# B&R Automation Studio project NAINV104C00R8L515F00 (part 27)

#### Local.var - Do Not Change!!!
```iecst
(*2020-09-10*)
(**)
(*Local Action, State & Status*)
VAR
	eAct : eHermesAction := HermesActIdle;
	eStat : eHermesAction := HermesActIdle;
	eMainStatus : eFBStatus := Idle;
	eStatus : eFBStatus := Idle;
	eStatus1 : eFBStatus := Idle;
	eStatus2 : eFBStatus := Idle;
	eStatus3 : eFBStatus := Idle;
	eStatus4 : eFBStatus := Idle;
	udiStatus : UDINT := 0;
	udiStatus1 : UDINT := 0;
	udiStatus2 : UDINT := 0;
	udiStatus3 : UDINT := 0;
	udiStatus4 : UDINT := 0;
	udiStatus5 : UDINT := 0;
	sStatTxt : STRING[200] := '';
	a_sStatText : ARRAY[0..50] OF STRING[200] := ['Idling','Background Starting Operations','Background Stopping Operations','Deleting Old Log File','Creating Directory','Writing Retain File','Reading Retain File','Saving Configuration',43('')];
END_VAR
(**)
(*Local Alarm*)
VAR
	tyAlmData : tyAlmDat;
	tyAlmData1 : tyAlmDat;
	tyAlmData2 : tyAlmDat;
	tyAlmData3 : tyAlmDat;
	tyAlmData4 : tyAlmDat;
	tyAlmData5 : tyAlmDat;
	tyInfoData : tyAlmDat;
	tyInfoData1 : tyAlmDat;
	tyInfoData2 : tyAlmDat;
	a_tyAlmText : ARRAY[10000..10199] OF tyAlmTxt := [(sAlmText:='Invalid Ident While Client Connecting',sRcyText:='Problem Occurred In The TCP/IP Connection. Check The Connection And Try To Reconnect.'),(sAlmText:='Setting Keep Alive Interval Time Error While Client Connecting',sRcyText:='Unable To Establish Connection Between Machine. Check For Setting And Resume Operation.'),(sAlmText:='Setting Keep Alive Idle Time Error While Client Connecting',sRcyText:='Unable To Establish Connection Between Machine. Check For Setting And Resume Operation.'),(sAlmText:='Setting Keep Alive Count Error While Client Connecting',sRcyText:='Unable To Establish Connection Between Machine. Check For Setting And Resume Operation.'),(sAlmText:='Setting Keep Alive Error While Client Connecting',sRcyText:='Unable To Establish Connection Between Machine. Check For Setting And Resume Operation.'),(sAlmText:='Setting Receive Buffer Error While Client Connecting',sRcyText:='Unable To Establish Connection Between Machine. Check For Setting And Resume Operation.'),(sAlmText:='Setting Send Buffer Error While Client Connecting',sRcyText:='Unable To Establish Connection Between Machine. Check For Setting And Resume Operation.'),(sAlmText:='Setting No Waiting Error While Client Connecting',sRcyText:='Unable To Establish Connection Between Machine. Check For Setting And Resume Operation.'),(sAlmText:='TCP Open Port Error While Client Connecting',sRcyText:='Problem Occurred In The TCP/IP Connection. Check The Connection And Try To Reconnect.'),(sAlmText:='Closing TCP Error While Client Connecting',sRcyText:='Problem Occurred In The TCP/IP Connection. Check The Connection And Try To Reconnect.'),(sAlmText:='Server Connection Failed While Client Connecting',sRcyText:='There Was A Problem Connecting To The Server. The Server May Not Exist or It is Unavailable At This Time. Check The Connection and Try Again.'),(sAlmText:='Ident In Used While Client Connecting',sRcyText:='Problem Occurred In The TCP/IP Connection. Check The Connection And Reconnect.'),(sAlmText:='Connect To Server Error While Client Connecting',sRcyText:='There Was A Problem Connecting To The Server. The Server May Not Exist or It is Unavailable At This Time. Check The Connection and Try Again.'),(sAlmText:='US Hermes Connection Lost',sRcyText:='Please Check Network Connection.'),(sAlmText:='Invalid Ident While Receiving Data',sRcyText:='Problem Occurred In The TCP/IP Connection. Check The Connection And Try To Reconnect.'),(sAlmText:='TCP Receive Data Error While Receiving Data',sRcyText:='Problem Occurred In The TCP/IP Connection. Check The Connection And Try To Reconnect.'),(sAlmText:='Receive ServiceDescription While Upstream In Not Connected State',sRcyText:='Receive Illegal Message.'),(sAlmText:='Receive BoardAvailable While Upstream In Not Connected State',sRcyText:='Receive Illegal Message.'),(sAlmText:='Receive RevokeBoardAvailable While Upstream In Not Connected State',sRcyText:='Receive Illegal Message.'),(sAlmText:='Receive MachineReady While Upstream In Not Connected State',sRcyText:='Receive Illegal Message.'),(sAlmText:='Receive RevokeMachineReady While Upstream In Not Connected State',sRcyText:='Receive Illegal Message.'),(sAlmText:='Receive StartTransport While Upstream In Not Connected State',sRcyText:='Receive Illegal Message.'),(sAlmText:='Receive StopTransport While Upstream In Not Connected State',sRcyText:='Receive Illegal Message.'),(sAlmText:='Receive TransportFinished While Upstream In Not Connected State',sRcyText:='Receive Illegal Message.'),(sAlmText:='Receive BoardForecast While Upstream In Not Connected State',sRcyText:='Receive Illegal Message.'),(sAlmText:='Receive BoardAvailable While Upstream In Service Description State',sRcyText:='Receive Illegal Message.'),(sAlmText:='Receive RevokeBoardAvailable While Upstream In Service Description State',sRcyText:='Receive Illegal Message.'),(sAlmText:='Receive MachineReady While Upstream In Service Description State',sRcyText:='Receive Illegal Message.'),(sAlmText:='Receive RevokeMachineReady While Upstream In Service Description State',sRcyText:='Receive Illegal Message.'),(sAlmText:='Receive StartTransport While Upstream In Service Description State',sRcyText:='Receive Illegal Message.'),(sAlmText:='Receive StopTransport While Upstream In Service Description State',sRcyText:='Receive Illegal Message.'),(sAlmText:='Receive TransportFinished While Upstream In Service Description State',sRcyText:='Receive Illegal Message.'),(sAlmText:='Receive BoardForecast While Upstream In Service Description State',sRcyText:='Receive Illegal Message.'),(sAlmText:='Receive ServiceDescription While Upstream In Not Available Not Ready State',sRcyText:='Receive Illegal Message.'),(sAlmText:='Receive RevokeBoardAvailable While Upstream In Not Available Not Ready State',sRcyText:='Receive Illegal Message.'),(sAlmText:='Receive MachineReady While Upstream In Not Available Not Ready State',sRcyText:='Receive Illegal Message.'),(sAlmText:='Receive RevokeMachineReady While Upstream In Not Available Not Ready State',sRcyText:='Receive Illegal Message.'),(sAlmText:='Receive StartTransport While Upstream In Not Available Not Ready State',sRcyText:='Receive Illegal Message.'),(sAlmText:='Receive StopTransport While Upstream In Not Available Not Ready State',sRcyText:='Receive Illegal Message.'),(sAlmText:='Receive TransportFinished While Upstream In Not Available Not Ready State',sRcyText:='Receive Illegal Message.'),(sAlmText:='Receive ServiceDescription While Upstream In Board Available State',sRcyText:='Receive Illegal Message.'),(sAlmText:='Receive BoardAvailable While Upstream In Board Available State',sRcyText:='Receive Illegal Message.'),(sAlmText:='Receive MachineReady While Upstream In Board Available State',sRcyText:='Receive Illegal Message.'),(sAlmText:='Receive RevokeMachineReady While Upstream In Board Available State',sRcyText:='Receive Illegal Message.'),(sAlmText:='Receive StartTransport While Upstream In Board Available State',sRcyText:='Receive Illegal Message.'),(sAlmText:='Receive StopTransport While Upstream In Board Available State',sRcyText:='Receive Illegal Message.'),(sAlmText:='Receive TransportFinished While Upstream In Board Available State',sRcyText:='Receive Illegal Message.'),(sAlmText:='Receive BoardForecast While Upstream In Board Available State',sRcyText:='Receive Illegal Message.'),(sAlmText:='Receive ServiceDescription While Upstream In Machine Ready State',sRcyText:='Receive Illegal Message.'),(sAlmText:='Receive RevokeBoardAvailable While Upstream In Machine Ready State',sRcyText:='Receive Illegal Message.'),(sAlmText:='Receive MachineReady While Upstream In Machine Ready State',sRcyText:='Receive Illegal Message.'),(sAlmText:='Receive RevokeMachineReady While Upstream In Machine Ready State',sRcyText:='Receive Illegal Message.'),(sAlmText:='Receive StartTransport While Upstream In Machine Ready State',sRcyText:='Receive Illegal Message.'),(sAlmText:='Receive StopTransport While Upstream In Machine Ready State',sRcyText:='Receive Illegal Message.'),(sAlmText:='Receive TransportFinished While Upstream In Machine Ready State',sRcyText:='Receive Illegal Message.'),(sAlmText:='Receive ServiceDescription While Upstream In Available And Ready State',sRcyText:='Receive Illegal Message.'),(sAlmText:='Receive BoardAvailable While Upstream In Available And Ready State',sRcyText:='Receive Illegal Message.'),(sAlmText:='Receive MachineReady While Upstream In Available And Ready State',sRcyText:='Receive Illegal Message.'),(sAlmText:='Receive RevokeMachineReady While Upstream In Available And Ready State',sRcyText:='Receive Illegal Message.'),(sAlmText:='Receive StartTransport While Upstream In Available And Ready State',sRcyText:='Receive Illegal Message.'),(sAlmText:='Receive StopTransport While Upstream In Available And Ready State',sRcyText:='Receive Illegal Message.'),(sAlmText:='Receive TransportFinished While Upstream In Available And Ready State',sRcyText:='Receive Illegal Message.'),(sAlmText:='Receive BoardForecast While Upstream In Available And Ready State',sRcyText:='Receive Illegal Message.'),(sAlmText:='Receive ServiceDescription While Upstream In Transporting State',sRcyText:='Receive Illegal Message.'),(sAlmText:='Receive Twice Board Available While Upstream In Transporting State',sRcyText:='Receive Illegal Message.'),(sAlmText:='Receive RevokeBoardAvailable Without BoardAvailable While Upstream In Transporting State',sRcyText:='Receive Illegal Message.'),(sAlmText:='Receive MachineReady While Upstream In Transporting State',sRcyText:='Receive Illegal Message.'),(sAlmText:='Receive RevokeMachineReady While Upstream In Transporting State',sRcyText:='Receive Illegal Message.'),(sAlmText:='Receive StartTransport While Upstream In Transporting State',sRcyText:='Receive Illegal Message.'),(sAlmText:='Receive StopTransport While Upstream In Transporting State',sRcyText:='Receive Illegal Message.'),(sAlmText:='Receive ServiceDescription While Upstream In Transport Finished State',sRcyText:='Receive Illegal Message.'),(sAlmText:='Receive BoardAvailable While Upstream In Transport Finished State',sRcyText:='Receive Illegal Message.'),(sAlmText:='Receive RevokeBoardAvailable While UpstreamWhile Upstream In Transport Finished State',sRcyText:='Receive Illegal Message.'),(sAlmText:='Receive MachineReady While Upstream In Transport Finished State',sRcyText:='Receive Illegal Message.'),(sAlmText:='Receive RevokeMachineReady While Upstream In Transport Finished State',sRcyText:='Receive Illegal Message.'),(sAlmText:='Receive StartTransport While Upstream In Transport Finished State',sRcyText:='Receive Illegal Message.'),(sAlmText:='Receive TransportFinished While Upstream In Transport Finished State',sRcyText:='Receive Illegal Message.'),(sAlmText:='Receive StopTransport While Upstream In Transport Finished State',sRcyText:='Receive Illegal Message.'),(sAlmText:='Receive BoardForecast While Upstream In Transport Finished State',sRcyText:='Receive Illegal Message.'),(sAlmText:='Receive ServiceDescription While Upstream In Transport Stopped State',sRcyText:='Receive Illegal Message.'),(sAlmText:='Receive Twice Board Available While Upstream In Transport Stopped State',sRcyText:='Receive Illegal Message.'),(sAlmText:='Receive RevokeBoardAvailable Without BoardAvailable While Upstream In Transport Stopped State',sRcyText:='Receive Illegal Message.'),(sAlmText:='Receive MachineReady While Upstream In Transport Stopped State',sRcyText:='Receive Illegal Message.'),(sAlmText:='Receive RevokeMachineReady While Upstream In Transport Stopped State',sRcyText:='Receive Illegal Message.'),(sAlmText:='Receive StartTransport While Upstream In Transport Stopped State',sRcyText:='Receive Illegal Message.'),(sAlmText:='Receive StopTransport While Upstream In Transport Stopped State',sRcyText:='Receive Illegal Message.'),(sAlmText:='LaneId Mismatch While Checking Service Description',sRcyText:='The LaneId Value Does Not Match. Change The Value And Resend The Value.'),(sAlmText:='MachineId Missing While Checking Service Description',sRcyText:='Missing Input Value For MachineId. Fill Up The Value And Resend.'),(sAlmText:='LandId Out Of Range While Checking Service Description',sRcyText:='LaneId Does Not Fall Within The Expected Range.'),(sAlmText:='LandId Missing While Checking Service Description',sRcyText:='Missing Input Value For LaneId. Fill Up The Value And Resend.'),(sAlmText:='Version Missing While Checking Service Description',sRcyText:='Missing Input Value For Version. Fill Up The Value And Resend.'),(sAlmText:='SupportedFeatures Missing While Checking Service Description',sRcyText:='Missing Input Value For SupportedFeatures. Fill Up The Value And Resend.'),(sAlmText:='NotificationCode Out Of Range While Checking Notification',sRcyText:='NotificationCode Does Not Fall Within The Expected Range.'),(sAlmText:='NotificationCode Missing While Checking Notification',sRcyText:='Missing Input Value For NotificationCode. Fill Up The Value And Resend.'),(sAlmText:='Severity Missing While Checking Notification',sRcyText:='Missing Input Value For Severity. Fill Up The Value And Resend.'),(sAlmText:='Description Missing While Checking Notification',sRcyText:='Missing Input Value For Description. Fill Up The Value And Resend.'),(sAlmText:='BoardId Missing While Checking Board Available',sRcyText:='Missing Input Value For BoardId. Fill Up The Value And Resend.'),(sAlmText:='BoardIdCreatedBy Missing While Checking Board Available',sRcyText:='Missing Input Value For BoardIdCreatedBy. Fill Up The Value And Resend.'),(sAlmText:='FailedBoard Missing While Checking Board Available',sRcyText:='Missing Input Value For FailedBoard. Fill Up The Value And Resend.'),(sAlmText:='FlippedBoard Missing While Checking Board Available',sRcyText:='Missing Input Value For FlippedBoard. Fill Up The Value And Resend.'),(sAlmText:='TransferState Missing While Checking Transport Finished',sRcyText:='Missing Input Value For TransferState. Fill Up The Value And Resend.'),(sAlmText:='BoardId Missing While Checking Transport Finished',sRcyText:='Missing Input Value For BoardId. Fill Up The Value And Resend.'),(sAlmText:='FailedBoard Missing While Checking Board Forecast',sRcyText:='Missing Input Value For FailedBoard. Fill Up The Value And Resend.'),(sAlmText:='FlippedBoard Missing While Checking Board Forecast',sRcyText:='Missing Input Value For FlippedBoard. Fill Up The Value And Resend.'),(sAlmText:='BoardId Mismatch While Checking Start Transport & Transport Finished',sRcyText:='The BoardId Value Does Not Match. Change The Value And Resend The Value.'),(sAlmText:='BoardId Missing While Checking Start Transport & Transport Finished',sRcyText:='Missing Input Value For BoardId. Fill Up The Value And Resend.'),(sAlmText:='Service Description Interchange Time Out',sRcyText:='Timeout Expired Before Operation Completed. Reset And Resume Operation.'),(sAlmText:='Transport Time Out',sRcyText:='Timeout Expired Before Operation Completed. Reset And Resume Operation.'),(sAlmText:='Input First Slot Is Invalid',sRcyText:='Invalid Input Value.'),(sAlmText:='Input Last Slot Is Invalid',sRcyText:='Invalid Input Value.'),(sAlmText:='Input Pitch Is Invalid',sRcyText:='Invalid Input Value.'),(sAlmText:='Input Slot To Slot Distance Is Invalid',sRcyText:='Invalid Input Value.'),(sAlmText:='Input Total Slot Is Invalid',sRcyText:='Invalid Input Value.'),(sAlmText:='Input Thickness Is Invalid',sRcyText:='Invalid Input Value.'),(sAlmText:='Input Top Clearance Height Is Invalid',sRcyText:='Invalid Input Value.'),(sAlmText:='Input Bottom Clearance Height Is Invalid',sRcyText:='Invalid Input Value.'),(sAlmText:='Recipe First Slot Value & Board Available Data Not Match With Same Product Type Id',sRcyText:='The Recipe First Slot Value & Board Available Data Value Does Not Match With Product Type ID. Change The Value And Resend The Value.'),(sAlmText:='Recipe Last Slot Value & Board Available Data Not Match With Same Product Type Id',sRcyText:='The Recipe Last Slot Value & Board Available Data Value Does Not Match With Product Type ID. Change The Value And Resend The Value.'),(sAlmText:='Recipe Pitch Value & Board Available Data Not Match With Same Product Type Id',sRcyText:='The Recipe Pitch Value & Board Available Data Value Does Not Match With Product Type ID. Change The Value And Resend The Value.'),(sAlmText:='Width Different With Same Product Type Id',sRcyText:='Width Does Not Match With Product Type ID. Change The Value And Resend The Value.'),(sAlmText:='Input First Slot Is Invalid',sRcyText:='Invalid Input Value.'),(sAlmText:='Input Last Slot Is Invalid',sRcyText:='Invalid Input Value.'),(sAlmText:='Input Pitch Is Invalid',sRcyText:='Invalid Input Value.'),(sAlmText:='Input Slot To Slot Distance Is Invalid',sRcyText:='Invalid Input Value.'),(sAlmText:='Input Total Slot Is Invalid',sRcyText:='Invalid Input Value.'),(sAlmText:='Input Thickness Is Invalid',sRcyText:='Invalid Input Value.'),(sAlmText:='Input Top Clearance Height Is Invalid',sRcyText:='Invalid Input Value.'),(sAlmText:='Input Bottom Clearance Height Is Invalid',sRcyText:='Invalid Input Value.'),(sAlmText:='Recipe First Slot Value & Board Available Data Not Match With Same Product Type Id',sRcyText:='The Recipe First Slot Value & Board Available Data Value Does Not Match With Product Type ID. Change The Value And Resend The Value.'),(sAlmText:='Recipe Last Slot Value & Board Available Data Not Match With Same Product Type Id',sRcyText:='The Recipe Last Slot Value & Board Available Data Value Does Not Match With Product Type ID. Change The Value And Resend The Value.'),(sAlmText:='Recipe Pitch Value & Board Available Data Not Match With Same Product Type Id',sRcyText:='The Recipe Pitch Value & Board Available Data Value Does Not Match With Product Type ID. Change The Value And Resend The Value.'),(sAlmText:='Width Different With Same Product Type Id',sRcyText:='Width Does Not Match With Product Type ID. Change The Value And Resend The Value.'),(sAlmText:='Check Alive Time Out',sRcyText:='Timeout Expired Before Operation Completed. Reset And Resume Operation.'),(sAlmText:='Waiting Check Alive Time Out',sRcyText:='Timeout Expired Before Operation Completed. Reset And Resume Operation.'),(sAlmText:='Check Alive Id Mismatch',sRcyText:='The Check Alive Id Value Does Not Match. Change The Value And Resend The Value.'),(sAlmText:='Board Available Request To Send From Upstream Hermes',sRcyText:='Sending Illegal Message.'),(sAlmText:='Revoke Board Available Request To Send From Upstream Hermes',sRcyText:='Sending Illegal Message.'),(sAlmText:='Transport Finished Request To Send From Upstream Hermes',sRcyText:='Sending Illegal Message.'),(sAlmText:='Set Configuration Request To Send From Upstream Hermes',sRcyText:='Sending Illegal Message.'),(sAlmText:='Get Configuration Request To Send From Upstream Hermes',sRcyText:='Sending Illegal Message.'),(sAlmText:='Current Configuration Request To Send From Upstream Hermes',sRcyText:='Sending Illegal Message.'),(sAlmText:='Board Forecast Request To Send From Upstream Hermes',sRcyText:='Sending Illegal Message.'),(sAlmText:='Send Board Info Request To Send From Upstream Hermes',sRcyText:='Sending Illegal Message.'),(sAlmText:='Invalid Ident While Sending Data',sRcyText:='Invalid Ident Value.'),(sAlmText:='TCP Retry Send Data Error While Sending Data',sRcyText:='Problem Occurred In The TCP/IP Connection. Check The Connection And Try To Reconnect.'),(sAlmText:='TCP Send Data Error',sRcyText:='Problem Occurred In The TCP/IP Connection. Check The Connection And Try To Reconnect.'),(sAlmText:='Invalid Ident While Closing TCP',sRcyText:='Invalid Ident Value.'),(sAlmText:='Closing TCP Error',sRcyText:='Problem Occurred In The TCP/IP Connection. Check The Connection And Try To Reconnect.'),(sAlmText:='File Open Error While Writing Log',sRcyText:='An Error Was Encountered While Trying To Open File. Please Contact Nutek For A Possible Solution.'),(sAlmText:='File Create Error While Writing Log',sRcyText:='An Error Was Encountered While Trying To Create File. Please Contact Nutek For A Possible Solution.'),(sAlmText:='Get File Info Error While Writing Log',sRcyText:='An Error Was Encountered While Getting File Info. Please Contact Nutek For A Possible Solution.'),(sAlmText:='File Write Error While Writing Log',sRcyText:='An Error Was Encountered While Trying To Write File. Please Contact Nutek For A Possible Solution.'),(sAlmText:='File Close Error While Writing Log',sRcyText:='An Error Was Encountered While Trying To Close File. Please Contact Nutek For A Possible Solution.'),(sAlmText:='Directory Does Not Exist While Writing Log',sRcyText:='The Directory Does Not Exist.Please Contact Nutek For A Possible Solution.'),(sAlmText:='Get Directory Info Error While Deleting Old Log',sRcyText:='An Error Was Encountered While Getting Directory Info. Please Contact Nutek For A Possible Solution.'),(sAlmText:='Directory Read Error While Deleting Old Log',sRcyText:='An Error Was Encountered While Reading Directory. Please Contact Nutek For A Possible Solution.'),(sAlmText:='File Delete Error While Deleting Old Log',sRcyText:='An Error Was Encountered While Trying To Delete File. Please Contact Nutek For A Possible Solution.'),(sAlmText:='Board Jam At Sensor After Transfer Interrupted',sRcyText:='Push Back Board To Upstream Machine'),(sAlmText:='Product Type Id Not Receive From Upstream',sRcyText:='Check Upstream Machine Whether Product Type Id Is Used.'),10((0)),(sAlmText:='New Recipe Not Found In Product Recipe List',sRcyText:='Create New Recipe In Product Setting.'),30((0))];
END_VAR
(**)
(*Local Output*)
VAR
	a_tyXMLTableDataBrdAvl : ARRAY[0..200] OF tyXMLTableDat;
	iXMLTableDataBrdAvlTtlIdx : INT;
	bConnected : BOOL;
	bHandshakeDone : BOOL;
	bBoardChkReq : BOOL;
	bAccDataReq : BOOL;
	bProcessBoardForecastId : BOOL;
	bBFAccDataReq : BOOL;
	bOverWriteSlt : BOOL;
	bBFOverWriteSlt : BOOL;
	bBFOverWriteWidth : BOOL;
	bOverWriteWidth : BOOL;
	sReqRecipeNm : STRING[254];
	diReqWidthInUM : DINT;
	diReqMinSltValue : DINT;
	diReqMaxSltValue : DINT;
	diReqPitch : DINT;
	bNotAvlNotRdy : BOOL;
	bUSRdy : BOOL;
	bDSRdy : BOOL;
	bUSGdRdy : BOOL;
	bDSGdRdy : BOOL;
	iAction : INT;
	bTransporting : BOOL;
	bStopTransport : BOOL;
	tyBoardAvailableRcv : tyHermesBoardAvailable;
	tyBoardAvailableReq : tyHermesBoardAvailable;
	bBlkUS : BOOL;
	bBABlkUS : BOOL;
	bBFBlkUS : BOOL;
	bManuallInsertLastZone : BOOL;
	bReverseRcvBlkUS : BOOL;
	sInternalSnd : STRING[65535];
	bRcvBoardInfoOk : BOOL;
	bRcvBoardInfoIncompl : BOOL;
	tySendBoardInfoAcc : tyHermesSendBoardInfo;
END_VAR
(**)
(*Local Input*)
VAR
	udiRstErr : UDINT := 0;
	bPrep : BOOL := TRUE;
	bEn : BOOL := TRUE;
	bDis : BOOL := FALSE;
	tyParam : tyHermesUSParam := (tSndAlive:=T#30s,tRcvAlive:=T#60s,iLaneID:=1,sHostAddress:='192.168.0.200',uiHostPort:=5000);
	sIPAddr : STRING[15] := '192.168.0.100';
	tyDTStructure : DTStructure := (year:=2019,month:=01,day:=05,wday:=05,hour:=21,minute:=28,second:=30,millisec:=123,microsec:=456);
	dtCurrDT : DATE_AND_TIME := DT#2019-02-23-12:30:50;
	bRdyRcv : BOOL := FALSE;
	bRdyTransport : BOOL := FALSE;
	bRcvCompl : BOOL := FALSE;
	bRcvInCompl : BOOL := FALSE;
	bRcvNotStart : BOOL := FALSE;
	bBAWidthEn : BOOL := TRUE; (*Board Available Check Width*)
	bBASltEn : BOOL := FALSE; (*Board Available Check Slot*)
	bBFWidthEn : BOOL := TRUE; (*Board Forecast Check Width*)
	bBFSltEn : BOOL := FALSE; (*Board Forecast Check Slot*)
	sMcId : STRING[80] := '';
	sInterfaceId : STRING[80] := '';
	sVersion : STRING[7] := '1.0.2';
	eFailedBoard : eHermesFailedBoard := HermesUnknownBoard;
	sRecipeNm : STRING[254] := '';
	diWidthInUM : DINT := 0;
	diMinSltValue : DINT := 0;
	diMaxSltValue : DINT := 0;
	diPitch : DINT := 0;
	diTtlSlt : DINT := 0;
	diSltToSltInUM : DINT := 0;
	udiSndBffrSize : UDINT := 65536;
	udiRcvBffrSize : UDINT := 65536;
	udiAliveIdleTimeInSec : UDINT := 5;
	tConnTimeOut : TIME := T#30s;
	diTransferInTO : DINT := 30000;
	bOpsRun : BOOL := FALSE;
	bInterruptSen : BOOL := FALSE;
	udiFileKeepDay : UDINT := 30;
	sProgNm : STRING[15] := 'USHermes';
	bNtSettingsLoadDone : BOOL := TRUE;
	bAccDataRdy : BOOL := FALSE;
	sRmtMcId : STRING[80];
	bRmtPrep : BOOL := FALSE;
	bRmtEn : BOOL := FALSE;
	bAccNewRcpCond : BOOL;
	sInfoMsg : STRING[200];
	sInfoMsg1 : STRING[200];
	sInfoMsg2 : STRING[200];
	bInternalUse : BOOL;
	sInternalRcv : STRING[65535];
	a_tyProdRcpList : ARRAY[1..c_udiProdRcpMax] OF tyProdRcpParam;
	tyProdRcpCurrRcp : tyProdRcpParam;
	bMcParamMnlAccData : BOOL;
	bUIAccData : BOOL;
END_VAR
(**)
(*Local*)
VAR
	bRstErr : BOOL;
	udiRstErrOld : UDINT;
	bInitDone : BOOL;
	bInitialDone : BOOL;
	bRun : BOOL;
	bStop : BOOL;
	bRstConnection : BOOL;
	bRstState : BOOL;
	udiTCPIdent : UDINT;
	udiXMLTableWriteIdx : UDINT;
	udiMsgSendBffr : UDINT;
	udiSndMsgLen : UDINT;
	sSnd : STRING[65535];
	sRcv : STRING[65535];
	a_tyXMLTableDataRcv : ARRAY[0..200] OF tyXMLTableDat;
	a_tyXMLTableDataSnd : ARRAY[0..200] OF tyXMLTableDat;
	a_eMsgSend : ARRAY[0..50] OF eHermesMsgType;
	tyMsgTypeRcv : tyHermesMsgType;
	tyCheckAliveSnd : tyHermesCheckAlive;
	tyCheckAlivePingSnd : tyHermesCheckAlive;
	tyCheckAlivePongSnd : tyHermesCheckAlive;
	tyCheckAliveRcv : tyHermesCheckAlive;
	tyCheckAlivePingRcv : tyHermesCheckAlive;
	tyCheckAlivePongRcv : tyHermesCheckAlive;
	tyServiceDescriptionSnd : tyHermesServiceDescription;
	tyServiceDescriptionRcv : tyHermesServiceDescription;
	tyNotificationSnd : tyHermesNotification;
	tyNotificationRcv : tyHermesNotification;
	tyBoardAvailableDummy : tyHermesBoardAvailable;
	tyBoardArrivedInfo : tyHermesBoardAvailable;
	tyMachineReady : tyHermesMachineReady;
	tyStartTransport : tyHermesStartTransport;
	tyStopTransport : tyHermesStopTransport;
	tyTransportFinished : tyHermesTransportFinished;
	tySetConfiguration : tyHermesSetConfiguration;
	tyCurrentConfiguration : tyHermesCurrentConfiguration;
	tyBoardForecastRcv : tyHermesBoardForecast;
	tyBoardForecastAcc : tyHermesBoardForecast;
	tyQueryBoardInfo : tyHermesQueryBoardInfo;
	tySendBoardInfoRcv : tyHermesSendBoardInfo;
	tyCommandRcv : tyHermesCommand;
	tyCommandSnd : tyHermesCommand;
	fbClntConnect : fbTCPClntConnect;
	fbRcv : fbTCPRcv;
	fbSend : fbTCPSnd;
	fbClose : fbTCPClose;
	fbParseXMLTable : fbHermesParseXMLTable;
	fbCheckAlive : fbHermesCheckAlive;
	fbCheckAliveSendPing : fbHermesCheckAliveSendPing;
	fbCheckAliveRcvPing : fbHermesCheckAliveRcvPing;
	fbSequenceUS : fbHermesSequenceUS;
	fbSequenceTO : fbHermesSequenceTO;
	fbGetSlt : fbHermesGetSlt;
	eStatOld : eHermesAction := HermesActIdle;
	tyParamOld : tyHermesUSParam;
	udiLogCntr : UDINT := 1;
	udiWriteLogCntr : UDINT := 1;
	a_sLogList : ARRAY[1..10] OF STRING[65535];
	sDT : STRING[80];
	dtCurrDTTemp : DATE_AND_TIME;
	fbFileAppend1 : fbFileFullAppend;
	fbFileOldDel1 : fbFileOldDel;
	iWriteLogStep : INT := 0;
	i : INT;
	usiBFAccDataStep : USINT;
	usiAccDataStep : USINT;
	bFeatureBoardForecast : BOOL;
	bAccDataMnl : BOOL;
	bStopTransportSnd : BOOL;
	tyCommandParam : tyHermesCommandParam;
	a_usiHermesCommandIdx : ARRAY[0..7] OF USINT;
	udiModuleNum : UDINT := 3101;
	bReplyMcRdyId : BOOL;
	bBrdForecastRcv : BOOL;
END_VAR
(*Reverse Trigger*)
VAR
	bProcessRouteMachine : BOOL;
	bTriggerRouteMachine : BOOL;
	bProcessRouteReversal : BOOL;
	bTriggerRouteReversal : BOOL;
	iGotoLane : INT;
	bManualRmvBrdCond : BOOL;
	bReverseDSSndBfWBrdID : BOOL;
	bTriggerUpdateRoute : BOOL;
	bNotifyRstReverseRcvGate : BOOL;
	fbRstReverseRcvGate : TON;
	fbRstReverseDSSndBF : TON;
	usidx : USINT;
	iMinDis : INT;
	bSwitchtoReverseReceive : BOOL;
	fbRstSndBF : TON;
	bStopTransportSent : BOOL;
	bBoardAvailableRcved : BOOL;
END_VAR
(*Insert your comment here.*)
VAR
	bManualRmvRoute : BOOL;
	bReturnRoute : BOOL;
	bNomRouteEn : BOOL;
	bProcessRouteEn : BOOL;
	bReverseReceiveRoute : BOOL;
	bReceiveReverseUSMcRdy : BOOL;
	bReverseSentRoute : BOOL;
END_VAR
(*QueryBoard Info*)
VAR
	sUITopBarcode : STRING[254];
	sUIBottomBarcode : STRING[254];
END_VAR
```

### USHermes2.var - Change By Project
```iecst
(*2020-09-10*)
(**)
(*Action & State & Status*)
VAR
	p_USHermes2Stat : UDINT;
	p_USHermes2Status : UDINT;
	p_USHermes2StatTxt : UDINT;
END_VAR
(**)
(*Alarm*)
VAR
	p_USHermes2AlmData : UDINT;
	p_USHermes2AlmData1 : UDINT;
	p_USHermes2AlmData2 : UDINT;
	p_USHermes2AlmData3 : UDINT;
	p_USHermes2AlmData4 : UDINT;
	p_USHermes2AlmData5 : UDINT;
	p_USHermes2InfoData : UDINT;
END_VAR
(**)
(*Output*)
VAR
	p_USHermes2TableDataBrdAvl : UDINT;
	p_USHermes2TableDataBrdAvlTtlIdx : UDINT;
	p_USHermes2Connected : UDINT;
	p_USHermes2HandshakeDone : UDINT;
	p_USHermes2AccDataReq : UDINT;
	p_USHermes2OverWriteSlt : UDINT;
	p_USHermes2OverWriteWidth : UDINT;
	p_USHermes2ReqRecipeNm : UDINT;
	p_USHermes2ReqWidthInUM : UDINT;
	p_USHermes2ReqMinSltValue : UDINT;
	p_USHermes2ReqMaxSltValue : UDINT;
	p_USHermes2ReqPitch : UDINT;
	p_USHermes2USRdy : UDINT;
	p_USHermes2DSRdy : UDINT;
	p_USHermes2USGdRdy : UDINT;
	p_USHermes2DSGdRdy : UDINT;
	p_USHermes2Transporting : UDINT;
	p_USHermes2StopTransport : UDINT;
	p_USHermes2BlkUS : UDINT;
	p_USHermes2InternalSnd : UDINT;
	p_USHermes2AccDataMnl : UDINT;
	p_USHermes2tyBoardAvailable : UDINT;
	p_USHermes2CommandParam : UDINT;
	p_USHermes2ReverseDSSendBFId : UDINT;
	p_USHermes2ProcessRouteTrigger : UDINT;
	p_USHermes2SwitchtoReverseRcv : UDINT;
	p_USHermes2StopTransportSnd : UDINT;
	p_USHermes2RcvBoardInfoOk : UDINT;
	p_USHermes2RcvbBoardInfoIncompl : UDINT;
	p_USHermes2BoardInfoData : UDINT;
	p_USHermes2BoardArrivedData : UDINT;
	p_USHermes2BrdForecastRcv : UDINT;
	p_USHermes2BoardAvailableRcved : UDINT;
	p_USHermes2StopTransportSent : UDINT;
	p_USHermes2StopTransportSentMsg : UDINT;
	p_USHermes2BrdForecast : UDINT;
END_VAR
```

### Program Logical/Hermes/USHermes2 (IEC) - 1.00.0 - NtHermes v5.00.0 , NtTCP v5.00.0 , NtMessage v5.00.0

#### InputRef.var
```iecst
(*2019-06-28*)
(**)
(*General*)
VAR
	p_eAct : REFERENCE TO eHermesAction;
	p_udiRstErr : REFERENCE TO UDINT;
	p_bPrep : REFERENCE TO BOOL;
	p_bEn : REFERENCE TO BOOL;
	p_bDis : REFERENCE TO BOOL;
END_VAR
(**)
(*Configuration*)
VAR
	p_tyParam : REFERENCE TO tyHermesUSParam;
	p_sIPAddr : REFERENCE TO STRING[15];
	p_tyDTStructure : REFERENCE TO DTStructure;
	p_dtCurrDT : REFERENCE TO DATE_AND_TIME;
END_VAR
(**)
(*Input*)
VAR
	p_bRdyRcv : REFERENCE TO BOOL;
	p_bRdyTransport : REFERENCE TO BOOL;
	p_bRcvCompl : REFERENCE TO BOOL;
	p_bRcvIncompl : REFERENCE TO BOOL;
	p_bRcvNotStart : REFERENCE TO BOOL;
	p_bBAWidthEn : REFERENCE TO BOOL; (*Board Available Check Width*)
	p_bBASltEn : REFERENCE TO BOOL; (*Board Available Check Slot*)
	p_bBFWidthEn : REFERENCE TO BOOL; (*Board Forecast Check Width*)
	p_bBFSltEn : REFERENCE TO BOOL; (*Board Forecast Check Slot*)
	p_sMcId : REFERENCE TO STRING[80];
	p_sInterfaceId : REFERENCE TO STRING[80];
	p_sVersion : REFERENCE TO STRING[7];
	p_eFailedBoard : REFERENCE TO eHermesFailedBoard;
	p_eFlippedBoard : REFERENCE TO eHermesFlippedBoard;
	p_sRecipeNm : REFERENCE TO STRING[254];
	p_diWidthInUM : REFERENCE TO DINT;
	p_diMinSltValue : REFERENCE TO DINT;
	p_diMaxSltValue : REFERENCE TO DINT;
	p_diPitch : REFERENCE TO DINT;
	p_diTtlSlt : REFERENCE TO DINT;
	p_diSltToSltInUM : REFERENCE TO DINT;
	p_udiSndBffrSize : REFERENCE TO UDINT;
	p_udiRcvBffrSize : REFERENCE TO UDINT;
	p_udiAliveIdleTimeInSec : REFERENCE TO UDINT;
	p_tConnTimeOut : REFERENCE TO TIME;
	p_diTransferInTO : REFERENCE TO DINT;
	p_bOpsRun : REFERENCE TO BOOL;
	p_bInterruptSen : REFERENCE TO BOOL;
	p_udiFileKeepDay : REFERENCE TO UDINT;
	p_sProgNm : REFERENCE TO STRING[15];
	p_bNtSettingsLoadDone : REFERENCE TO BOOL;
	p_bAccDataRdy : REFERENCE TO BOOL;
	p_sRmtMcId : REFERENCE TO STRING[80];
	p_bRmtPrep : REFERENCE TO BOOL;
	p_bRmtEn : REFERENCE TO BOOL;
	p_bSvyPrep : REFERENCE TO BOOL;
	p_bSvyEn : REFERENCE TO BOOL;
	p_bAccNewRcpCond : REFERENCE TO BOOL;
	p_sInfoMsg : REFERENCE TO STRING[200];
	p_sInfoMsg1 : REFERENCE TO STRING[200];
	p_sInfoMsg2 : REFERENCE TO STRING[200];
	p_bInternalUse : REFERENCE TO BOOL;
	p_sInternalRcv : REFERENCE TO STRING[65535];
	p_tyCommand : REFERENCE TO tyHermesCommand;
	pa_tyProdRcpList : REFERENCE TO ARRAY[1..c_udiProdRcpMax] OF tyProdRcpParam;
	p_tyProdRcpCurrRcp : REFERENCE TO tyProdRcpParam;
	p_bMcParamMnlAccData : REFERENCE TO BOOL;
	p_bUIAccData : REFERENCE TO BOOL;
	p_bConvHvBrd : REFERENCE TO BOOL;
	p_bQueryBoardInfo : REFERENCE TO BOOL;
	p_bManualInsertZoneHvBrd : REFERENCE TO BOOL;
	p_bManualInsertEndSen : REFERENCE TO BOOL;
	pa_tyHermesDSParam : REFERENCE TO ARRAY[0..c_diHermesConfigMaxIdx] OF tyHermesDSParam;
END_VAR
(*Hermes Route*)
VAR
	p_bProcessRouteEn : REFERENCE TO BOOL;
	p_bManualRmvRoute : REFERENCE TO BOOL;
	p_bReturnRoute : REFERENCE TO BOOL;
	p_bNomRouteEn : REFERENCE TO BOOL;
	p_bReverseReceiveRoute : REFERENCE TO BOOL;
	p_bReceiveReverseUSMcRdy : REFERENCE TO BOOL;
	p_tyDSHermesCurrBASnd : REFERENCE TO tyHermesBoardAvailable;
	p_bHermesSwitchtoRvrseTransport : REFERENCE TO BOOL;
END_VAR
(*QueryBoardInfo
*)
VAR
	p_bTransportFinished : REFERENCE TO BOOL;
	p_sTopBarcode : REFERENCE TO STRING[254];
	p_sBottomBarcode : REFERENCE TO STRING[254];
END_VAR
```

#### Local.var
```iecst
(*2020-09-10*)
(**)
(*Local Action, State & Status*)
VAR
	eAct : eHermesAction := HermesActIdle;
	eStat : eHermesAction := HermesActIdle;
	eMainStatus : eFBStatus := Idle;
	eStatus : eFBStatus := Idle;
	eStatus1 : eFBStatus := Idle;
	eStatus2 : eFBStatus := Idle;
	eStatus3 : eFBStatus := Idle;
	eStatus4 : eFBStatus := Idle;
	udiStatus : UDINT := 0;
	udiStatus1 : UDINT := 0;
	udiStatus2 : UDINT := 0;
	udiStatus3 : UDINT := 0;
	udiStatus4 : UDINT := 0;
	udiStatus5 : UDINT := 0;
	sStatTxt : STRING[200] := '';
	a_sStatText : ARRAY[0..50] OF STRING[200] := ['Idling','Background Starting Operations','Background Stopping Operations','Deleting Old Log File','Creating Directory','Writing Retain File','Reading Retain File','Saving Configuration',43('')];
END_VAR
(**)
(*Local Alarm*)
VAR
	tyAlmData : tyAlmDat;
	tyAlmData1 : tyAlmDat;
	tyAlmData2 : tyAlmDat;
	tyAlmData3 : tyAlmDat;
	tyAlmData4 : tyAlmDat;
	tyAlmData5 : tyAlmDat;
	tyInfoData : tyAlmDat;
	tyInfoData1 : tyAlmDat;
	tyInfoData2 : tyAlmDat;
	a_tyAlmText : ARRAY[10000..10199] OF tyAlmTxt := [(sAlmText:='Invalid Ident While Client Connecting',sRcyText:='Problem Occurred In The TCP/IP Connection. Check The Connection And Try To Reconnect.'),(sAlmText:='Setting Keep Alive Interval Time Error While Client Connecting',sRcyText:='Unable To Establish Connection Between Machine. Check For Setting And Resume Operation.'),(sAlmText:='Setting Keep Alive Idle Time Error While Client Connecting',sRcyText:='Unable To Establish Connection Between Machine. Check For Setting And Resume Operation.'),(sAlmText:='Setting Keep Alive Count Error While Client Connecting',sRcyText:='Unable To Establish Connection Between Machine. Check For Setting And Resume Operation.'),(sAlmText:='Setting Keep Alive Error While Client Connecting',sRcyText:='Unable To Establish Connection Between Machine. Check For Setting And Resume Operation.'),(sAlmText:='Setting Receive Buffer Error While Client Connecting',sRcyText:='Unable To Establish Connection Between Machine. Check For Setting And Resume Operation.'),(sAlmText:='Setting Send Buffer Error While Client Connecting',sRcyText:='Unable To Establish Connection Between Machine. Check For Setting And Resume Operation.'),(sAlmText:='Setting No Waiting Error While Client Connecting',sRcyText:='Unable To Establish Connection Between Machine. Check For Setting And Resume Operation.'),(sAlmText:='TCP Open Port Error While Client Connecting',sRcyText:='Problem Occurred In The TCP/IP Connection. Check The Connection And Try To Reconnect.'),(sAlmText:='Closing TCP Error While Client Connecting',sRcyText:='Problem Occurred In The TCP/IP Connection. Check The Connection And Try To Reconnect.'),(sAlmText:='Server Connection Failed While Client Connecting',sRcyText:='There Was A Problem Connecting To The Server. The Server May Not Exist or It is Unavailable At This Time. Check The Connection and Try Again.'),(sAlmText:='Ident In Used While Client Connecting',sRcyText:='Problem Occurred In The TCP/IP Connection. Check The Connection And Reconnect.'),(sAlmText:='Connect To Server Error While Client Connecting',sRcyText:='There Was A Problem Connecting To The Server. The Server May Not Exist or It is Unavailable At This Time. Check The Connection and Try Again.'),(sAlmText:='US Hermes Connection Lost',sRcyText:='Please Check Network Connection.'),(sAlmText:='Invalid Ident While Receiving Data',sRcyText:='Problem Occurred In The TCP/IP Connection. Check The Connection And Try To Reconnect.'),(sAlmText:='TCP Receive Data Error While Receiving Data',sRcyText:='Problem Occurred In The TCP/IP Connection. Check The Connection And Try To Reconnect.'),(sAlmText:='Receive ServiceDescription While Upstream In Not Connected State',sRcyText:='Receive Illegal Message.'),(sAlmText:='Receive BoardAvailable While Upstream In Not Connected State',sRcyText:='Receive Illegal Message.'),(sAlmText:='Receive RevokeBoardAvailable While Upstream In Not Connected State',sRcyText:='Receive Illegal Message.'),(sAlmText:='Receive MachineReady While Upstream In Not Connected State',sRcyText:='Receive Illegal Message.'),(sAlmText:='Receive RevokeMachineReady While Upstream In Not Connected State',sRcyText:='Receive Illegal Message.'),(sAlmText:='Receive StartTransport While Upstream In Not Connected State',sRcyText:='Receive Illegal Message.'),(sAlmText:='Receive StopTransport While Upstream In Not Connected State',sRcyText:='Receive Illegal Message.'),(sAlmText:='Receive TransportFinished While Upstream In Not Connected State',sRcyText:='Receive Illegal Message.'),(sAlmText:='Receive BoardForecast While Upstream In Not Connected State',sRcyText:='Receive Illegal Message.'),(sAlmText:='Receive BoardAvailable While Upstream In Service Description State',sRcyText:='Receive Illegal Message.'),(sAlmText:='Receive RevokeBoardAvailable While Upstream In Service Description State',sRcyText:='Receive Illegal Message.'),(sAlmText:='Receive MachineReady While Upstream In Service Description State',sRcyText:='Receive Illegal Message.'),(sAlmText:='Receive RevokeMachineReady While Upstream In Service Description State',sRcyText:='Receive Illegal Message.'),(sAlmText:='Receive StartTransport While Upstream In Service Description State',sRcyText:='Receive Illegal Message.'),(sAlmText:='Receive StopTransport While Upstream In Service Description State',sRcyText:='Receive Illegal Message.'),(sAlmText:='Receive TransportFinished While Upstream In Service Description State',sRcyText:='Receive Illegal Message.'),(sAlmText:='Receive BoardForecast While Upstream In Service Description State',sRcyText:='Receive Illegal Message.'),(sAlmText:='Receive ServiceDescription While Upstream In Not Available Not Ready State',sRcyText:='Receive Illegal Message.'),(sAlmText:='Receive RevokeBoardAvailable While Upstream In Not Available Not Ready State',sRcyText:='Receive Illegal Message.'),(sAlmText:='Receive MachineReady While Upstream In Not Available Not Ready State',sRcyText:='Receive Illegal Message.'),(sAlmText:='Receive RevokeMachineReady While Upstream In Not Available Not Ready State',sRcyText:='Receive Illegal Message.'),(sAlmText:='Receive StartTransport While Upstream In Not Available Not Ready State',sRcyText:='Receive Illegal Message.'),(sAlmText:='Receive StopTransport While Upstream In Not Available Not Ready State',sRcyText:='Receive Illegal Message.'),(sAlmText:='Receive TransportFinished While Upstream In Not Available Not Ready State',sRcyText:='Receive Illegal Message.'),(sAlmText:='Receive ServiceDescription While Upstream In Board Available State',sRcyText:='Receive Illegal Message.'),(sAlmText:='Receive BoardAvailable While Upstream In Board Available State',sRcyText:='Receive Illegal Message.'),(sAlmText:='Receive MachineReady While Upstream In Board Available State',sRcyText:='Receive Illegal Message.'),(sAlmText:='Receive RevokeMachineReady While Upstream In Board Available State',sRcyText:='Receive Illegal Message.'),(sAlmText:='Receive StartTransport While Upstream In Board Available State',sRcyText:='Receive Illegal Message.'),(sAlmText:='Receive StopTransport While Upstream In Board Available State',sRcyText:='Receive Illegal Message.'),(sAlmText:='Receive TransportFinished While Upstream In Board Available State',sRcyText:='Receive Illegal Message.'),(sAlmText:='Receive BoardForecast While Upstream In Board Available State',sRcyText:='Receive Illegal Message.'),(sAlmText:='Receive ServiceDescription While Upstream In Machine Ready State',sRcyText:='Receive Illegal Message.'),(sAlmText:='Receive RevokeBoardAvailable While Upstream In Machine Ready State',sRcyText:='Receive Illegal Message.'),(sAlmText:='Receive MachineReady While Upstream In Machine Ready State',sRcyText:='Receive Illegal Message.'),(sAlmText:='Receive RevokeMachineReady While Upstream In Machine Ready State',sRcyText:='Receive Illegal Message.'),(sAlmText:='Receive StartTransport While Upstream In Machine Ready State',sRcyText:='Receive Illegal Message.'),(sAlmText:='Receive StopTransport While Upstream In Machine Ready State',sRcyText:='Receive Illegal Message.'),(sAlmText:='Receive TransportFinished While Upstream In Machine Ready State',sRcyText:='Receive Illegal Message.'),(sAlmText:='Receive ServiceDescription While Upstream In Available And Ready State',sRcyText:='Receive Illegal Message.'),(sAlmText:='Receive BoardAvailable While Upstream In Available And Ready State',sRcyText:='Receive Illegal Message.'),(sAlmText:='Receive MachineReady While Upstream In Available And Ready State',sRcyText:='Receive Illegal Message.'),(sAlmText:='Receive RevokeMachineReady While Upstream In Available And Ready State',sRcyText:='Receive Illegal Message.'),(sAlmText:='Receive StartTransport While Upstream In Available And Ready State',sRcyText:='Receive Illegal Message.'),(sAlmText:='Receive StopTransport While Upstream In Available And Ready State',sRcyText:='Receive Illegal Message.'),(sAlmText:='Receive TransportFinished While Upstream In Available And Ready State',sRcyText:='Receive Illegal Message.'),(sAlmText:='Receive BoardForecast While Upstream In Available And Ready State',sRcyText:='Receive Illegal Message.'),(sAlmText:='Receive ServiceDescription While Upstream In Transporting State',sRcyText:='Receive Illegal Message.'),(sAlmText:='Receive Twice Board Available While Upstream In Transporting State',sRcyText:='Receive Illegal Message.'),(sAlmText:='Receive RevokeBoardAvailable Without BoardAvailable While Upstream In Transporting State',sRcyText:='Receive Illegal Message.'),(sAlmText:='Receive MachineReady While Upstream In Transporting State',sRcyText:='Receive Illegal Message.'),(sAlmText:='Receive RevokeMachineReady While Upstream In Transporting State',sRcyText:='Receive Illegal Message.'),(sAlmText:='Receive StartTransport While Upstream In Transporting State',sRcyText:='Receive Illegal Message.'),(sAlmText:='Receive StopTransport While Upstream In Transporting State',sRcyText:='Receive Illegal Message.'),(sAlmText:='Receive ServiceDescription While Upstream In Transport Finished State',sRcyText:='Receive Illegal Message.'),(sAlmText:='Receive BoardAvailable While Upstream In Transport Finished State',sRcyText:='Receive Illegal Message.'),(sAlmText:='Receive RevokeBoardAvailable While UpstreamWhile Upstream In Transport Finished State',sRcyText:='Receive Illegal Message.'),(sAlmText:='Receive MachineReady While Upstream In Transport Finished State',sRcyText:='Receive Illegal Message.'),(sAlmText:='Receive RevokeMachineReady While Upstream In Transport Finished State',sRcyText:='Receive Illegal Message.'),(sAlmText:='Receive StartTransport While Upstream In Transport Finished State',sRcyText:='Receive Illegal Message.'),(sAlmText:='Receive TransportFinished While Upstream In Transport Finished State',sRcyText:='Receive Illegal Message.'),(sAlmText:='Receive StopTransport While Upstream In Transport Finished State',sRcyText:='Receive Illegal Message.'),(sAlmText:='Receive BoardForecast While Upstream In Transport Finished State',sRcyText:='Receive Illegal Message.'),(sAlmText:='Receive ServiceDescription While Upstream In Transport Stopped State',sRcyText:='Receive Illegal Message.'),(sAlmText:='Receive Twice Board Available While Upstream In Transport Stopped State',sRcyText:='Receive Illegal Message.'),(sAlmText:='Receive RevokeBoardAvailable Without BoardAvailable While Upstream In Transport Stopped State',sRcyText:='Receive Illegal Message.'),(sAlmText:='Receive MachineReady While Upstream In Transport Stopped State',sRcyText:='Receive Illegal Message.'),(sAlmText:='Receive RevokeMachineReady While Upstream In Transport Stopped State',sRcyText:='Receive Illegal Message.'),(sAlmText:='Receive StartTransport While Upstream In Transport Stopped State',sRcyText:='Receive Illegal Message.'),(sAlmText:='Receive StopTransport While Upstream In Transport Stopped State',sRcyText:='Receive Illegal Message.'),(sAlmText:='LaneId Mismatch While Checking Service Description',sRcyText:='The LaneId Value Does Not Match. Change The Value And Resend The Value.'),(sAlmText:='MachineId Missing While Checking Service Description',sRcyText:='Missing Input Value For MachineId. Fill Up The Value And Resend.'),(sAlmText:='LandId Out Of Range While Checking Service Description',sRcyText:='LaneId Does Not Fall Within The Expected Range.'),(sAlmText:='LandId Missing While Checking Service Description',sRcyText:='Missing Input Value For LaneId. Fill Up The Value And Resend.'),(sAlmText:='Version Missing While Checking Service Description',sRcyText:='Missing Input Value For Version. Fill Up The Value And Resend.'),(sAlmText:='SupportedFeatures Missing While Checking Service Description',sRcyText:='Missing Input Value For SupportedFeatures. Fill Up The Value And Resend.'),(sAlmText:='NotificationCode Out Of Range While Checking Notification',sRcyText:='NotificationCode Does Not Fall Within The Expected Range.'),(sAlmText:='NotificationCode Missing While Checking Notification',sRcyText:='Missing Input Value For NotificationCode. Fill Up The Value And Resend.'),(sAlmText:='Severity Missing While Checking Notification',sRcyText:='Missing Input Value For Severity. Fill Up The Value And Resend.'),(sAlmText:='Description Missing While Checking Notification',sRcyText:='Missing Input Value For Description. Fill Up The Value And Resend.'),(sAlmText:='BoardId Missing While Checking Board Available',sRcyText:='Missing Input Value For BoardId. Fill Up The Value And Resend.'),(sAlmText:='BoardIdCreatedBy Missing While Checking Board Available',sRcyText:='Missing Input Value For BoardIdCreatedBy. Fill Up The Value And Resend.'),(sAlmText:='FailedBoard Missing While Checking Board Available',sRcyText:='Missing Input Value For FailedBoard. Fill Up The Value And Resend.'),(sAlmText:='FlippedBoard Missing While Checking Board Available',sRcyText:='Missing Input Value For FlippedBoard. Fill Up The Value And Resend.'),(sAlmText:='TransferState Missing While Checking Transport Finished',sRcyText:='Missing Input Value For TransferState. Fill Up The Value And Resend.'),(sAlmText:='BoardId Missing While Checking Transport Finished',sRcyText:='Missing Input Value For BoardId. Fill Up The Value And Resend.'),(sAlmText:='FailedBoard Missing While Checking Board Forecast',sRcyText:='Missing Input Value For FailedBoard. Fill Up The Value And Resend.'),(sAlmText:='FlippedBoard Missing While Checking Board Forecast',sRcyText:='Missing Input Value For FlippedBoard. Fill Up The Value And Resend.'),(sAlmText:='BoardId Mismatch While Checking Start Transport & Transport Finished',sRcyText:='The BoardId Value Does Not Match. Change The Value And Resend The Value.'),(sAlmText:='BoardId Missing While Checking Start Transport & Transport Finished',sRcyText:='Missing Input Value For BoardId. Fill Up The Value And Resend.'),(sAlmText:='Service Description Interchange Time Out',sRcyText:='Timeout Expired Before Operation Completed. Reset And Resume Operation.'),(sAlmText:='Transport Time Out',sRcyText:='Timeout Expired Before Operation Completed. Reset And Resume Operation.'),(sAlmText:='Input First Slot Is Invalid',sRcyText:='Invalid Input Value.'),(sAlmText:='Input Last Slot Is Invalid',sRcyText:='Invalid Input Value.'),(sAlmText:='Input Pitch Is Invalid',sRcyText:='Invalid Input Value.'),(sAlmText:='Input Slot To Slot Distance Is Invalid',sRcyText:='Invalid Input Value.'),(sAlmText:='Input Total Slot Is Invalid',sRcyText:='Invalid Input Value.'),(sAlmText:='Input Thickness Is Invalid',sRcyText:='Invalid Input Value.'),(sAlmText:='Input Top Clearance Height Is Invalid',sRcyText:='Invalid Input Value.'),(sAlmText:='Input Bottom Clearance Height Is Invalid',sRcyText:='Invalid Input Value.'),(sAlmText:='Recipe First Slot Value & Board Available Data Not Match With Same Product Type Id',sRcyText:='The Recipe First Slot Value & Board Available Data Value Does Not Match With Product Type ID. Change The Value And Resend The Value.'),(sAlmText:='Recipe Last Slot Value & Board Available Data Not Match With Same Product Type Id',sRcyText:='The Recipe Last Slot Value & Board Available Data Value Does Not Match With Product Type ID. Change The Value And Resend The Value.'),(sAlmText:='Recipe Pitch Value & Board Available Data Not Match With Same Product Type Id',sRcyText:='The Recipe Pitch Value & Board Available Data Value Does Not Match With Product Type ID. Change The Value And Resend The Value.'),(sAlmText:='Width Different With Same Product Type Id',sRcyText:='Width Does Not Match With Product Type ID. Change The Value And Resend The Value.'),(sAlmText:='Input First Slot Is Invalid',sRcyText:='Invalid Input Value.'),(sAlmText:='Input Last Slot Is Invalid',sRcyText:='Invalid Input Value.'),(sAlmText:='Input Pitch Is Invalid',sRcyText:='Invalid Input Value.'),(sAlmText:='Input Slot To Slot Distance Is Invalid',sRcyText:='Invalid Input Value.'),(sAlmText:='Input Total Slot Is Invalid',sRcyText:='Invalid Input Value.'),(sAlmText:='Input Thickness Is Invalid',sRcyText:='Invalid Input Value.'),(sAlmText:='Input Top Clearance Height Is Invalid',sRcyText:='Invalid Input Value.'),(sAlmText:='Input Bottom Clearance Height Is Invalid',sRcyText:='Invalid Input Value.'),(sAlmText:='Recipe First Slot Value & Board Available Data Not Match With Same Product Type Id',sRcyText:='The Recipe First Slot Value & Board Available Data Value Does Not Match With Product Type ID. Change The Value And Resend The Value.'),(sAlmText:='Recipe Last Slot Value & Board Available Data Not Match With Same Product Type Id',sRcyText:='The Recipe Last Slot Value & Board Available Data Value Does Not Match With Product Type ID. Change The Value And Resend The Value.'),(sAlmText:='Recipe Pitch Value & Board Available Data Not Match With Same Product Type Id',sRcyText:='The Recipe Pitch Value & Board Available Data Value Does Not Match With Product Type ID. Change The Value And Resend The Value.'),(sAlmText:='Width Different With Same Product Type Id',sRcyText:='Width Does Not Match With Product Type ID. Change The Value And Resend The Value.'),(sAlmText:='Check Alive Time Out',sRcyText:='Timeout Expired Before Operation Completed. Reset And Resume Operation.'),(sAlmText:='Waiting Check Alive Time Out',sRcyText:='Timeout Expired Before Operation Completed. Reset And Resume Operation.'),(sAlmText:='Check Alive Id Mismatch',sRcyText:='The Check Alive Id Value Does Not Match. Change The Value And Resend The Value.'),(sAlmText:='Board Available Request To Send From Upstream Hermes',sRcyText:='Sending Illegal Message.'),(sAlmText:='Revoke Board Available Request To Send From Upstream Hermes',sRcyText:='Sending Illegal Message.'),(sAlmText:='Transport Finished Request To Send From Upstream Hermes',sRcyText:='Sending Illegal Message.'),(sAlmText:='Set Configuration Request To Send From Upstream Hermes',sRcyText:='Sending Illegal Message.'),(sAlmText:='Get Configuration Request To Send From Upstream Hermes',sRcyText:='Sending Illegal Message.'),(sAlmText:='Current Configuration Request To Send From Upstream Hermes',sRcyText:='Sending Illegal Message.'),(sAlmText:='Board Forecast Request To Send From Upstream Hermes',sRcyText:='Sending Illegal Message.'),(sAlmText:='Send Board Info Request To Send From Upstream Hermes',sRcyText:='Sending Illegal Message.'),(sAlmText:='Invalid Ident While Sending Data',sRcyText:='Invalid Ident Value.'),(sAlmText:='TCP Retry Send Data Error While Sending Data',sRcyText:='Problem Occurred In The TCP/IP Connection. Check The Connection And Try To Reconnect.'),(sAlmText:='TCP Send Data Error',sRcyText:='Problem Occurred In The TCP/IP Connection. Check The Connection And Try To Reconnect.'),(sAlmText:='Invalid Ident While Closing TCP',sRcyText:='Invalid Ident Value.'),(sAlmText:='Closing TCP Error',sRcyText:='Problem Occurred In The TCP/IP Connection. Check The Connection And Try To Reconnect.'),(sAlmText:='File Open Error While Writing Log',sRcyText:='An Error Was Encountered While Trying To Open File. Please Contact Nutek For A Possible Solution.'),(sAlmText:='File Create Error While Writing Log',sRcyText:='An Error Was Encountered While Trying To Create File. Please Contact Nutek For A Possible Solution.'),(sAlmText:='Get File Info Error While Writing Log',sRcyText:='An Error Was Encountered While Getting File Info. Please Contact Nutek For A Possible Solution.'),(sAlmText:='File Write Error While Writing Log',sRcyText:='An Error Was Encountered While Trying To Write File. Please Contact Nutek For A Possible Solution.'),(sAlmText:='File Close Error While Writing Log',sRcyText:='An Error Was Encountered While Trying To Close File. Please Contact Nutek For A Possible Solution.'),(sAlmText:='Directory Does Not Exist While Writing Log',sRcyText:='The Directory Does Not Exist.Please Contact Nutek For A Possible Solution.'),(sAlmText:='Get Directory Info Error While Deleting Old Log',sRcyText:='An Error Was Encountered While Getting Directory Info. Please Contact Nutek For A Possible Solution.'),(sAlmText:='Directory Read Error While Deleting Old Log',sRcyText:='An Error Was Encountered While Reading Directory. Please Contact Nutek For A Possible Solution.'),(sAlmText:='File Delete Error While Deleting Old Log',sRcyText:='An Error Was Encountered While Trying To Delete File. Please Contact Nutek For A Possible Solution.'),(sAlmText:='Board Jam At Sensor After Transfer Interrupted',sRcyText:='Push Back Board To Upstream Machine'),(sAlmText:='Product Type Id Not Receive From Upstream',sRcyText:='Check Upstream Machine Whether Product Type Id Is Used.'),10((0)),(sAlmText:='New Recipe Not Found In Product Recipe List',sRcyText:='Create New Recipe In Product Setting.'),30((0))];
END_VAR
(**)
(*Local Output*)
VAR
	a_tyXMLTableDataBrdAvl : ARRAY[0..200] OF tyXMLTableDat;
	iXMLTableDataBrdAvlTtlIdx : INT;
	bConnected : BOOL;
	bHandshakeDone : BOOL;
	bBoardChkReq : BOOL;
	bAccDataReq : BOOL;
	bProcessBoardForecastId : BOOL;
	bBFAccDataReq : BOOL;
	bOverWriteSlt : BOOL;
	bBFOverWriteSlt : BOOL;
	bBFOverWriteWidth : BOOL;
	bOverWriteWidth : BOOL;
	sReqRecipeNm : STRING[254];
	diReqWidthInUM : DINT;
	diReqMinSltValue : DINT;
	diReqMaxSltValue : DINT;
	diReqPitch : DINT;
	bNotAvlNotRdy : BOOL;
	bUSRdy : BOOL;
	bDSRdy : BOOL;
	bUSGdRdy : BOOL;
	bDSGdRdy : BOOL;
	iAction : INT;
	bTransporting : BOOL;
	bStopTransport : BOOL;
	tyBoardAvailableRcv : tyHermesBoardAvailable;
	tyBoardAvailableReq : tyHermesBoardAvailable;
	bBlkUS : BOOL;
	bBABlkUS : BOOL;
	bBFBlkUS : BOOL;
	bManuallInsertLastZone : BOOL;
	bReverseRcvBlkUS : BOOL;
	sInternalSnd : STRING[65535];
	bRcvBoardInfoOk : BOOL;
	bRcvBoardInfoIncompl : BOOL;
	tySendBoardInfoAcc : tyHermesSendBoardInfo;
END_VAR
(**)
(*Local Input*)
VAR
	udiRstErr : UDINT := 0;
	bPrep : BOOL := TRUE;
	bEn : BOOL := TRUE;
	bDis : BOOL := FALSE;
	tyParam : tyHermesUSParam := (tSndAlive:=T#30s,tRcvAlive:=T#60s,iLaneID:=1,sHostAddress:='192.168.0.200',uiHostPort:=5000);
	sIPAddr : STRING[15] := '192.168.0.100';
	tyDTStructure : DTStructure := (year:=2019,month:=01,day:=05,wday:=05,hour:=21,minute:=28,second:=30,millisec:=123,microsec:=456);
	dtCurrDT : DATE_AND_TIME := DT#2019-02-23-12:30:50;
	bRdyRcv : BOOL := FALSE;
	bRdyTransport : BOOL := FALSE;
	bRcvCompl : BOOL := FALSE;
	bRcvInCompl : BOOL := FALSE;
	bRcvNotStart : BOOL := FALSE;
	bBAWidthEn : BOOL := TRUE; (*Board Available Check Width*)
	bBASltEn : BOOL := FALSE; (*Board Available Check Slot*)
	bBFWidthEn : BOOL := TRUE; (*Board Forecast Check Width*)
	bBFSltEn : BOOL := FALSE; (*Board Forecast Check Slot*)
	sMcId : STRING[80] := '';
	sInterfaceId : STRING[80] := '';
	sVersion : STRING[7] := '1.0.2';
	eFailedBoard : eHermesFailedBoard := HermesUnknownBoard;
	sRecipeNm : STRING[254] := '';
	diWidthInUM : DINT := 0;
	diMinSltValue : DINT := 0;
	diMaxSltValue : DINT := 0;
	diPitch : DINT := 0;
	diTtlSlt : DINT := 0;
	diSltToSltInUM : DINT := 0;
	udiSndBffrSize : UDINT := 65536;
	udiRcvBffrSize : UDINT := 65536;
	udiAliveIdleTimeInSec : UDINT := 5;
	tConnTimeOut : TIME := T#30s;
	diTransferInTO : DINT := 30000;
	bOpsRun : BOOL := FALSE;
	bInterruptSen : BOOL := FALSE;
	udiFileKeepDay : UDINT := 30;
	sProgNm : STRING[15] := 'USHermes';
	bNtSettingsLoadDone : BOOL := TRUE;
	bAccDataRdy : BOOL := FALSE;
	sRmtMcId : STRING[80];
	bRmtPrep : BOOL := FALSE;
	bRmtEn : BOOL := FALSE;
	bAccNewRcpCond : BOOL;
	sInfoMsg : STRING[200];
	sInfoMsg1 : STRING[200];
	sInfoMsg2 : STRING[200];
	bInternalUse : BOOL;
	sInternalRcv : STRING[65535];
	a_tyProdRcpList : ARRAY[1..c_udiProdRcpMax] OF tyProdRcpParam;
	tyProdRcpCurrRcp : tyProdRcpParam;
	bMcParamMnlAccData : BOOL;
	bUIAccData : BOOL;
END_VAR
(**)
(*Local*)
VAR
	bRstErr : BOOL;
	udiRstErrOld : UDINT;
	bInitDone : BOOL;
	bInitialDone : BOOL;
	bRun : BOOL;
	bStop : BOOL;
	bRstConnection : BOOL;
	bRstState : BOOL;
	udiTCPIdent : UDINT;
	udiXMLTableWriteIdx : UDINT;
	udiMsgSendBffr : UDINT;
	udiSndMsgLen : UDINT;
	sSnd : STRING[65535];
	sRcv : STRING[65535];
	a_tyXMLTableDataRcv : ARRAY[0..200] OF tyXMLTableDat;
	a_tyXMLTableDataSnd : ARRAY[0..200] OF tyXMLTableDat;
	a_eMsgSend : ARRAY[0..50] OF eHermesMsgType;
	tyMsgTypeRcv : tyHermesMsgType;
	tyCheckAliveSnd : tyHermesCheckAlive;
	tyCheckAlivePingSnd : tyHermesCheckAlive;
	tyCheckAlivePongSnd : tyHermesCheckAlive;
	tyCheckAliveRcv : tyHermesCheckAlive;
	tyCheckAlivePingRcv : tyHermesCheckAlive;
	tyCheckAlivePongRcv : tyHermesCheckAlive;
	tyServiceDescriptionSnd : tyHermesServiceDescription;
	tyServiceDescriptionRcv : tyHermesServiceDescription;
	tyNotificationSnd : tyHermesNotification;
	tyNotificationRcv : tyHermesNotification;
	tyBoardAvailableDummy : tyHermesBoardAvailable;
	tyBoardArrivedInfo : tyHermesBoardAvailable;
	tyMachineReady : tyHermesMachineReady;
	tyStartTransport : tyHermesStartTransport;
	tyStopTransport : tyHermesStopTransport;
	tyTransportFinished : tyHermesTransportFinished;
	tySetConfiguration : tyHermesSetConfiguration;
	tyCurrentConfiguration : tyHermesCurrentConfiguration;
	tyBoardForecastRcv : tyHermesBoardForecast;
	tyBoardForecastAcc : tyHermesBoardForecast;
	tyQueryBoardInfo : tyHermesQueryBoardInfo;
	tySendBoardInfoRcv : tyHermesSendBoardInfo;
	tyCommandRcv : tyHermesCommand;
	tyCommandSnd : tyHermesCommand;
	fbClntConnect : fbTCPClntConnect;
	fbRcv : fbTCPRcv;
	fbSend : fbTCPSnd;
	fbClose : fbTCPClose;
	fbParseXMLTable : fbHermesParseXMLTable;
	fbCheckAlive : fbHermesCheckAlive;
	fbCheckAliveSendPing : fbHermesCheckAliveSendPing;
	fbCheckAliveRcvPing : fbHermesCheckAliveRcvPing;
	fbSequenceUS : fbHermesSequenceUS;
	fbSequenceTO : fbHermesSequenceTO;
	fbGetSlt : fbHermesGetSlt;
	eStatOld : eHermesAction := HermesActIdle;
	tyParamOld : tyHermesUSParam;
	udiLogCntr : UDINT := 1;
	udiWriteLogCntr : UDINT := 1;
	a_sLogList : ARRAY[1..10] OF STRING[65535];
	sDT : STRING[80];
	dtCurrDTTemp : DATE_AND_TIME;
	fbFileAppend1 : fbFileFullAppend;
	fbFileOldDel1 : fbFileOldDel;
	iWriteLogStep : INT := 0;
	i : INT;
	usiBFAccDataStep : USINT;
	usiAccDataStep : USINT;
	bFeatureBoardForecast : BOOL;
	bAccDataMnl : BOOL;
	bStopTransportSnd : BOOL;
	tyCommandParam : tyHermesCommandParam;
	a_usiHermesCommandIdx : ARRAY[0..7] OF USINT;
	udiModuleNum : UDINT := 3101;
	bReplyMcRdyId : BOOL;
	bBrdForecastRcv : BOOL;
END_VAR
(*Reverse Trigger*)
VAR
	bProcessRouteMachine : BOOL;
	bTriggerRouteMachine : BOOL;
	bProcessRouteReversal : BOOL;
	bTriggerRouteReversal : BOOL;
	iGotoLane : INT;
	bManualRmvBrdCond : BOOL;
	bReverseDSSndBfWBrdID : BOOL;
	bTriggerUpdateRoute : BOOL;
	bNotifyRstReverseRcvGate : BOOL;
	fbRstReverseRcvGate : TON;
	fbRstReverseDSSndBF : TON;
	usidx : USINT;
	iMinDis : INT;
	bSwitchtoReverseReceive : BOOL;
	fbRstSndBF : TON;
	bStopTransportSent : BOOL;
	bBoardAvailableRcved : BOOL;
END_VAR
(*Insert your comment here.*)
VAR
	bManualRmvRoute : BOOL;
	bReturnRoute : BOOL;
	bNomRouteEn : BOOL;
	bProcessRouteEn : BOOL;
	bReverseReceiveRoute : BOOL;
	bReceiveReverseUSMcRdy : BOOL;
	bReverseSentRoute : BOOL;
	bSwitchtoReverseRcv : BOOL;
END_VAR
(*QueryBoard Info*)
VAR
	sUITopBarcode : STRING[254];
	sUIBottomBarcode : STRING[254];
END_VAR
```

#### Act_Action.st
```iecst
(** 2019-03-25 **)
ACTION Act_Action:

	//Reset Error
	IF (eStatus = Error) AND bRstErr THEN
		p_eAct	:= HermesActIdle;
		eStat	:= HermesActIdle;
	END_IF

	//Set p_eAct
	IF eStatus = Idle OR eStatus = Done THEN //OR eStatus = Busy
		eStat	:= p_eAct;
	END_IF

END_ACTION
```

#### Act_Alarm1.st
```iecst
(** 2021-08-01 **)
ACTION Act_Alarm1: //General

	//Error
	IF EDGEPOS(eStatus1 = Error) THEN

		tyAlmData1.sProgNm		:= p_sProgNm;
		tyAlmData1.udiCode		:= udiStatus1;
		tyAlmData1.eSeverity	:= AlmSeverityError;
		tyAlmData1.udiRunTime	:= tyAlmData1.udiRunTime + 1;
		tyAlmData1.bAlm			:= TRUE;
		tyAlmData1.udiModuleNum := udiModuleNum;
		g_sUSHermesProgNm		:= p_sProgNm;

		//Get Error Message
		IF tyAlmData1.udiCode < 10000 OR tyAlmData1.udiCode > 10199 THEN
			tyAlmData1.sAlmMsg	:= 'Unknown';
			tyAlmData1.sRcyMsg	:= 'Unknown';
		ELSE
			tyAlmData1.sAlmMsg	:= a_tyAlmText[tyAlmData1.udiCode].sAlmText;
			tyAlmData1.sRcyMsg	:= a_tyAlmText[tyAlmData1.udiCode].sRcyText;
		END_IF

		sStatTxt	:= tyAlmData1.sAlmMsg;

	ELSIF bRstErr AND (tyAlmData1.udiCode <> 0) THEN

		tyAlmData1.udiCode		:= 0;
		tyAlmData1.eSeverity	:= AlmSeverityNA;
		tyAlmData1.sAlmMsg		:= '';
		tyAlmData1.sRcyMsg		:= '';
		tyAlmData1.bAlm			:= FALSE;
		sStatTxt	:= a_sStatText[eStat];

	END_IF

END_ACTION
```

#### Act_Alarm5.st
```iecst
(** 2022-12-20 **)
ACTION Act_Alarm5: //Not Connected Warning

	//Warning
	IF ((bConnected = FALSE) AND (p_eLinkMcParamUSCommMod= McSetCommModHermes)) THEN

		tyAlmData5.sProgNm		:= p_sProgNm;
		tyAlmData5.udiCode		:= udiStatus5;
		tyAlmData5.eSeverity	:= AlmSeverityWarning;
		tyAlmData5.udiRunTime	:= tyAlmData5.udiRunTime + 1;
		tyAlmData5.bWarning		:= TRUE;
		tyAlmData5.udiModuleNum := udiModuleNum;
		g_sUSHermesProgNm		:= p_sProgNm;

		//Get Warning Message
		IF tyAlmData5.udiCode < 10000 OR tyAlmData5.udiCode > 10199 THEN
			tyAlmData5.sAlmMsg	:= 'Unknown';
			tyAlmData5.sRcyMsg	:= 'Unknown';
		ELSE
			tyAlmData5.sAlmMsg	:= a_tyAlmText[tyAlmData5.udiCode].sAlmText;
			tyAlmData5.sRcyMsg	:= a_tyAlmText[tyAlmData5.udiCode].sRcyText;
		END_IF

		sStatTxt	:= tyAlmData5.sAlmMsg;

	ELSIF (bConnected AND (tyAlmData5.udiCode <> 0)) OR (p_eLinkMcParamUSCommMod = McSetCommModSMEMA)  THEN

		tyAlmData5.udiCode			:= 0;
		tyAlmData5.eSeverity		:= AlmSeverityNA;
		tyAlmData5.sAlmMsg			:= '';
		tyAlmData5.sRcyMsg			:= '';
		tyAlmData5.bWarning		   := FALSE;

		sStatTxt	:= a_sStatText[eStat];

	END_IF

END_ACTION
```

#### Act_Background.st
```iecst
(** 2019-06-10 **)
ACTION Act_Background:
	Act_Background_Info;
	IF bRun = TRUE THEN
		IF udiTCPIdent = 0 THEN
			IF p_bInternalUse = FALSE THEN
				Act_Background_TCPConnect;

				tyParamOld	:= p_tyParam;
			ELSE
				udiTCPIdent	:= 1;
			END_IF

		ELSE
			IF bRstConnection = FALSE THEN
				Act_Background_TCPRcv;

				Act_Background_NotificationRcv;

				Act_Background_IllegalMsg;
				Act_Background_ChkParamRcv;
				Act_Background_CmpParamRcv;

				IF bHandshakeDone = TRUE THEN
					IF (p_tyParam.tSndAlive <> T#0s) AND (p_tyParam.tRcvAlive <> T#0s) THEN
						IF tyServiceDescriptionRcv.tyData.tySupportedFeatures.bFeatureCheckAliveResponse = TRUE AND p_tyParam.bFeatureCheckAliveResponse = TRUE THEN
							Act_Background_ChkAliveSendPing;
							Act_Background_ChkAliveRcvPing;
						ELSE
							Act_Background_ChkAlive;
						END_IF
					ELSE
						fbCheckAlive(bEn := FALSE);
						fbCheckAliveSendPing(bEn := FALSE);
						fbCheckAliveRcvPing(bEn := FALSE);
					END_IF
				END_IF
				Act_Background_BoardForecast;
				//Act_Background_BoardAvailableChk;
				Act_Background_RequestedBoardChk;
				//Act_Background_Route;
				Act_Background_Sequence;
				Act_Background_SequenceTO;
				Act_Background_Err;

				Act_Background_ProcessData;
				Act_Background_QueryBoardInfo;

				Act_Background_Command;

				Act_Background_ChgConfig;

				Act_Background_TCPSend;

				Act_Background_Log;

			ELSE
				Act_Background_TCPClose;

			END_IF

		END_IF

		Act_Background_Stop;

	END_IF

	IF EDGENEG(bRun) OR EDGENEG(udiTCPIdent = 0) THEN
		//Reset
		fbClntConnect(bEn := FALSE);

		bConnected	:= bRun;
	END_IF

	IF EDGENEG(bRun) OR EDGENEG(udiTCPIdent <> 0) THEN
		fbRcv(bEn := FALSE);
		fbSequenceUS(bEn := FALSE);
		fbSequenceTO(bEn := FALSE);
		fbCheckAlive(bEn := FALSE);
		fbCheckAliveSendPing(bEn := FALSE);
		fbCheckAliveRcvPing(bEn := FALSE);
		fbSend(bEn := FALSE);
		fbClose(bEn := FALSE);

		fbFileAppend1(bEn := FALSE);
		iWriteLogStep	:= 0;

		bConnected		    := FALSE;
		bHandshakeDone	    := FALSE;
		bBlkUS			    := FALSE;
		bBABlkUS			:= FALSE;
		bBFBlkUS			:= FALSE;
		bManuallInsertLastZone	:= FALSE;
		bAccDataReq		    := FALSE;
		bBFAccDataReq	    := FALSE;
		bOverWriteSlt    	:= FALSE;
		bOverWriteWidth	    := FALSE;
		bBFOverWriteSlt	    := FALSE;
		bBFOverWriteWidth	:= FALSE;
		bRstConnection    	:= FALSE;
		bRstState	    	:= FALSE;
		bUSRdy	    		:= FALSE;
		bDSRdy		    	:= FALSE;
		bTransporting    	:= FALSE;
		bStopTransport   	:= FALSE;

		memset(ADR(tyMsgTypeRcv) , 0 , SIZEOF(tyMsgTypeRcv));
		memset(ADR(a_eMsgSend) , 0 , SIZEOF(a_eMsgSend));
		udiMsgSendBffr	:= 0;
	END_IF

	//Reset Error
	IF (eStatus1 = Error) AND bRstErr THEN
		eStatus1	:= Idle;
		udiStatus1	:= 0;

		fbClntConnect(bEn := FALSE);
		fbRcv(bEn := FALSE);
		fbSequenceUS(bEn := FALSE);
		fbSend(bEn := FALSE);
		fbClose(bEn := FALSE);
		fbCheckAlive(bEn := FALSE);
		fbCheckAliveSendPing(bEn := FALSE);
		fbCheckAliveRcvPing(bEn := FALSE);
		fbSequenceTO(bEn := FALSE);

		fbFileAppend1(bEn := FALSE);
		iWriteLogStep	:= 0;

		bConnected		    := FALSE;
		bHandshakeDone	    := FALSE;
		bBlkUS			    := FALSE;
		bBABlkUS			:= FALSE;
		bBFBlkUS			:= FALSE;
		bManuallInsertLastZone	:= FALSE;
		bAccDataReq		    := FALSE;
		bBFAccDataReq	    := FALSE;
		bOverWriteSlt    	:= FALSE;
		bOverWriteWidth	    := FALSE;
		bBFOverWriteSlt	    := FALSE;
		bBFOverWriteWidth	:= FALSE;
		bRstConnection    	:= FALSE;
		bRstState	    	:= FALSE;
		bUSRdy	    		:= FALSE;
		bDSRdy		    	:= FALSE;
		bTransporting    	:= FALSE;
		bStopTransport   	:= FALSE;
		bBoardChkReq		:= FALSE; //Added

		memset(ADR(tyMsgTypeRcv) , 0 , SIZEOF(tyMsgTypeRcv));
		memset(ADR(a_eMsgSend) , 0 , SIZEOF(a_eMsgSend));
		udiMsgSendBffr	:= 0;
	END_IF

	IF (eStatus2 = Error) AND bRstErr THEN
		eStatus2	:= Idle;
		udiStatus2	:= 0;

		fbSequenceTO(bEn := FALSE);

	END_IF

	IF (eStatus3 = Error) AND bRstErr THEN
		eStatus3	:= Idle;
		udiStatus3	:= 0;

		fbFileAppend1(bEn := FALSE);
		iWriteLogStep	:= 0;
	END_IF

	IF (eStatus4 = Error) AND bRstErr THEN
		eStatus4	:= Idle;
		udiStatus4	:= 0;
	END_IF

	Act_Background_AccData;
	//Act_Background_BFAccData;

END_ACTION
```

#### Act_Background_AccData.st
```iecst
(** 2021-08-01 **)
ACTION Act_Background_AccData: //Accept BoardAvailable Data from Upstream

	CASE usiAccDataStep OF
		0:
			//Request Accept Data
			IF bBoardChkReq AND eMainStatus <> Error AND bAccDataReq = TRUE THEN //bUSRdy = TRUE
				usiAccDataStep	:= 1;
			END_IF

		1:
			//Manual Accept Data Check
			IF bAccDataReq = TRUE THEN
				IF p_bMcParamMnlAccData = TRUE THEN
					bAccDataMnl	:= TRUE;

					tyInfoData.sProgNm		:= p_sProgNm;
					tyInfoData.udiCode		:= 10000;
					tyInfoData.eSeverity	:= AlmSeverityInfo;
					tyInfoData.sAlmMsg		:= p_sInfoMsg;

					IF p_bUIAccData = TRUE THEN
						bAccDataMnl		:= FALSE;
						usiAccDataStep	:= 2;
					END_IF
				ELSE
					bAccDataMnl		:= FALSE;
					usiAccDataStep	:= 2;
				END_IF
			ELSE
				bAccDataMnl		:= FALSE;
				usiAccDataStep	:= 4;
			END_IF

		2:
			IF bAccDataReq = TRUE THEN
				IF p_bAccNewRcpCond = TRUE THEN //In Auto Mode, and empty
					usiAccDataStep	:= 3;
				ELSE
					//Info Message
					tyInfoData.sProgNm		:= p_sProgNm;
					tyInfoData.udiCode		:= 10000;
					tyInfoData.eSeverity	:= AlmSeverityInfo;
					tyInfoData.sAlmMsg		:= p_sInfoMsg;
				END_IF
			ELSE
				usiAccDataStep	:= 4;
			END_IF

		3:
			//Sync Recipe
			IF bOverWriteWidth = TRUE OR bOverWriteSlt = TRUE THEN

				//Accept New Recipe Width
				IF bOverWriteWidth = TRUE THEN
					p_tyProdRcpCurrRcp.diWidthInUM	:= diReqWidthInUM;
				END_IF

				//Accept New Recipe Slot
				IF bOverWriteSlt = TRUE THEN
					diReqMaxSltValue;
					diReqMinSltValue;
					diReqPitch;
				END_IF

			ELSE

				//Accept New Recipe Name
				FOR i := 1 TO 2000 DO
					IF sReqRecipeNm = pa_tyProdRcpList[i].sRcpNm THEN
						p_tyProdRcpCurrRcp	:= pa_tyProdRcpList[i];
						EXIT;
					END_IF
				END_FOR

				IF i > 2000 THEN
					//Recipe Not Exist
					eStatus4	:= Error;
					udiStatus4	:= 10169;	//New Recipe Not Found In Product Recipe List

					fHermesAddOneMsgSend(ADR(a_eMsgSend) , ADR(udiMsgSendBffr) , HermesMsgTypeNotification);

					tyNotificationSnd.tyAvl.bSeverity			:= TRUE;
					tyNotificationSnd.tyAvl.bNotificationCode	:= TRUE;
					tyNotificationSnd.tyAvl.bDescription		:= TRUE;
					tyNotificationSnd.tyData.eSeverity			:= HermesSeverityError;
					tyNotificationSnd.tyData.iNotificationCode	:= UDINT_TO_INT(udiStatus4);
					tyNotificationSnd.tyData.sDescription		:= a_tyAlmText[udiStatus4].sAlmText;

				END_IF

			END_IF

			usiAccDataStep	:= 4;

		4:
			//Clear Info Message
			tyInfoData.sProgNm		:= '';
			tyInfoData.udiCode		:= 0;
			tyInfoData.eSeverity	:= AlmSeverityNA;
			tyInfoData.sAlmMsg		:= '';

			usiAccDataStep	:= 0;

	END_CASE

END_ACTION
```

#### Act_Background_BFAccData.st
```iecst
(** 2021-08-01 **)
ACTION Act_Background_BFAccData: //Accept BoardForecast Data from Upstream

	CASE usiBFAccDataStep OF
		0:
			//Request Accept Data
			IF bProcessBoardForecastId = TRUE AND eMainStatus <> Error AND bBFAccDataReq = TRUE THEN
				usiBFAccDataStep	:= 1;
			END_IF

		1:
			//Manual Accept Data Check
			IF bBFAccDataReq = TRUE THEN
				IF p_bMcParamMnlAccData = TRUE THEN
					bAccDataMnl	:= TRUE; //use bAccDataMnl instead of bBFAccDataMnl

					tyInfoData.sProgNm		:= p_sProgNm;
					tyInfoData.udiCode		:= 10000;
					tyInfoData.eSeverity	:= AlmSeverityInfo;
					tyInfoData.sAlmMsg		:= p_sInfoMsg;

					IF p_bUIAccData = TRUE THEN
						bAccDataMnl		:= FALSE;
						usiBFAccDataStep	:= 2;
					END_IF
				ELSE
					bAccDataMnl		:= FALSE;
					usiBFAccDataStep	:= 2;
				END_IF
			ELSE
				bAccDataMnl		:= FALSE;
				usiBFAccDataStep	:= 4;
			END_IF

		2:
			IF bBFAccDataReq = TRUE THEN
				IF p_bAccNewRcpCond = TRUE THEN //In Auto Mode, and empty
					usiBFAccDataStep	:= 3;
				ELSE
					//Info Message
					tyInfoData.sProgNm		:= p_sProgNm;
					tyInfoData.udiCode		:= 10000;
					tyInfoData.eSeverity	:= AlmSeverityInfo;
					tyInfoData.sAlmMsg		:= p_sInfoMsg;
				END_IF
			ELSE
				usiBFAccDataStep	:= 4;
			END_IF

		3:
			//Sync Recipe
			IF bBFOverWriteWidth = TRUE OR bBFOverWriteSlt = TRUE THEN

				//Accept New Recipe Width
				IF bBFOverWriteWidth = TRUE THEN
					p_tyProdRcpCurrRcp.diWidthInUM	:= diReqWidthInUM;
				END_IF

				//Accept New Recipe Slot
				IF bBFOverWriteSlt = TRUE THEN
					diReqMaxSltValue;
					diReqMinSltValue;
					diReqPitch;
				END_IF

			ELSE

				//Accept New Recipe Name
				FOR i := 1 TO 2000 DO
					IF sReqRecipeNm = pa_tyProdRcpList[i].sRcpNm THEN
						p_tyProdRcpCurrRcp	:= pa_tyProdRcpList[i];
						EXIT;
					END_IF
				END_FOR

				IF i > 2000 THEN
					//Recipe Not Exist
					eStatus4	:= Error;
					udiStatus4	:= 10169;	//New Recipe Not Found In Product Recipe List

					fHermesAddOneMsgSend(ADR(a_eMsgSend) , ADR(udiMsgSendBffr) , HermesMsgTypeNotification);

					tyNotificationSnd.tyAvl.bSeverity			:= TRUE;
					tyNotificationSnd.tyAvl.bNotificationCode	:= TRUE;
					tyNotificationSnd.tyAvl.bDescription		:= TRUE;
					tyNotificationSnd.tyData.eSeverity			:= HermesSeverityError;
					tyNotificationSnd.tyData.iNotificationCode	:= 6; //BoreForecast Error
					tyNotificationSnd.tyData.sDescription		:= a_tyAlmText[udiStatus4].sAlmText;

				END_IF

			END_IF

			usiBFAccDataStep	:= 4;

		4:
			//Clear Info Message
			tyInfoData.sProgNm		:= '';
			tyInfoData.udiCode		:= 0;
			tyInfoData.eSeverity	:= AlmSeverityNA;
			tyInfoData.sAlmMsg		:= '';
			usiBFAccDataStep	:= 0;
			bReplyMcRdyId           := TRUE; //add
			bProcessBoardForecastId := FALSE; //add
	END_CASE

END_ACTION
```

#### Act_Background_BoardAvailableChk.st
```iecst
(** 2019-04-11 **)
ACTION Act_Background_BoardAvailableChk:

//	IF eStatus2 <> Error  THEN
//		                                                                                  //ADD
//		IF (p_bAccDataRdy = TRUE) AND (bTransporting = FALSE) AND (p_bOpsRun = TRUE) THEN // AND p_bUIInsertBrdPrep = FALSE  THEN
//
//			bAccDataReq		:= FALSE;
//			bBABlkUS		:= FALSE;
//			bOverWriteSlt	:= FALSE;
//			bOverWriteWidth	:= FALSE;
//
//			IF p_tyParam.bCmpTypeId = TRUE THEN	//"Compare Type ID" Ticked
//
//				IF tyBoardAvailableRcv.tyAvl.bProductTypeId = TRUE THEN	//Check if there is Product Type Id in B.A msg
//
//					IF tyBoardAvailableRcv.tyData.sProductTypeId <> p_sRecipeNm THEN	//Product Type Id Different
//
//						bAccDataReq	    := TRUE;	//Require To Load New Recipe
//						bBABlkUS		:= TRUE;
//
//						sReqRecipeNm	:= tyBoardAvailableRcv.tyData.sProductTypeId;
//						diReqWidthInUM	:= REAL_TO_DINT(tyBoardAvailableRcv.tyData.rWidth * 1000);
//
//					ELSE	//Product Type Id Same (After accepted or Originally same)
//
//						IF p_tyParam.bCmpParam = TRUE THEN	//"Compare Param" Ticked
//							IF tyBoardAvailableRcv.tyAvl.bThickness AND tyBoardAvailableRcv.tyAvl.bTopClearanceHeight AND tyBoardAvailableRcv.tyAvl.bBottomClearanceHeight AND p_bBASltEn THEN	//Camparing Slot Parameters if p_bBASltEn = TRUE
//								udiStatus2	:= fHermesCmpSlt(tyBoardAvailableRcv.tyData.eFlippedBoard , tyBoardAvailableRcv.tyData.rThickness , tyBoardAvailableRcv.tyData.rTopClearanceHeight , tyBoardAvailableRcv.tyData.rBottomClearanceHeight , p_diMinSltValue , p_diMaxSltValue , p_diPitch , p_diSltToSltInUM , p_diTtlSlt);
//
//								IF udiStatus2 <> 0 THEN
//
//									bBABlkUS	:= TRUE;
//
//									eStatus2	:= Error;
//
//									IF udiStatus2 = 2914 THEN
//										udiStatus2	:= 10108;	//Input First Slot Is Invalid
//									ELSIF udiStatus2 = 2915 THEN
//										udiStatus2	:= 10109;	//Input Last Slot Is Invalid
//									ELSIF udiStatus2 = 2916 THEN
//										udiStatus2	:= 10110;	//Input Pitch Is Invalid
//									ELSIF udiStatus2 = 2917 THEN
//										udiStatus2	:= 10111;	//Input Slot To Slot Distance Is Invalid
//									ELSIF udiStatus2 = 2918 THEN
//										udiStatus2	:= 10112;	//Input Total Slot Is Invalid
//									ELSIF udiStatus2 = 2919 THEN
//										udiStatus2	:= 10113;	//Input Thickness Is Invalid
//									ELSIF udiStatus2 = 2920 THEN
//										udiStatus2	:= 10114;	//Input Top Clearance Height Is Invalid
//									ELSIF udiStatus2 = 2921 THEN
//										udiStatus2	:= 10115;	//Input Bottom Clearance Height Is Invalid
//									ELSIF udiStatus2 = 2922 THEN
//										udiStatus2	:= 10116;	//Recipe First Slot Value & Board Available Data Not Match With Same Product Type Id
//									ELSIF udiStatus2 = 2923 THEN
//										udiStatus2	:= 10117;	//Recipe Last Slot Value & Board Available Data Not Match With Same Product Type Id
//									ELSIF udiStatus2 = 2924 THEN
//										udiStatus2	:= 10118;	//Recipe Pitch Value & Board Available Data Not Match With Same Product Type Id
//									END_IF
//
//									fHermesAddOneMsgSend(ADR(a_eMsgSend) , ADR(udiMsgSendBffr) , HermesMsgTypeNotification);
//
//									tyNotificationSnd.tyAvl.bSeverity			:= TRUE;
//									tyNotificationSnd.tyAvl.bNotificationCode	:= TRUE;
//									tyNotificationSnd.tyAvl.bDescription		:= TRUE;
//									tyNotificationSnd.tyData.eSeverity			:= HermesSeverityError;
//									tyNotificationSnd.tyData.iNotificationCode	:= UDINT_TO_INT(udiStatus2);
//									tyNotificationSnd.tyData.sDescription		:= a_tyAlmText[udiStatus2].sAlmText;
//
//								END_IF
//							END_IF
//
//							IF tyBoardAvailableRcv.tyAvl.bWidth AND p_bBAWidthEn THEN	//Comparing Width Parameter if p_bBAWidthEn = TRUE
//								IF REAL_TO_DINT(tyBoardAvailableRcv.tyData.rWidth * 1000) <> p_diWidthInUM THEN
//
//									bBABlkUS	:= TRUE;
//
//									eStatus2	:= Error;
//									udiStatus2	:= 10119;	//Width Different With Same Product Type Id
//
//									fHermesAddOneMsgSend(ADR(a_eMsgSend) , ADR(udiMsgSendBffr) , HermesMsgTypeNotification);
//
//									tyNotificationSnd.tyAvl.bSeverity			:= TRUE;
//									tyNotificationSnd.tyAvl.bNotificationCode	:= TRUE;
//									tyNotificationSnd.tyAvl.bDescription		:= TRUE;
//									tyNotificationSnd.tyData.eSeverity			:= HermesSeverityError;
//									tyNotificationSnd.tyData.iNotificationCode	:= UDINT_TO_INT(udiStatus2);
//									tyNotificationSnd.tyData.sDescription		:= a_tyAlmText[udiStatus2].sAlmText;
//
//								END_IF
//							END_IF
//
//						END_IF
//
//					END_IF
//
//				ELSE
//
//					eStatus2	:= Error;
//					udiStatus2	:= 10158;	//Product Type Id Not Receive From Upstream
//
//					fHermesAddOneMsgSend(ADR(a_eMsgSend) , ADR(udiMsgSendBffr) , HermesMsgTypeNotification);
//
//					tyNotificationSnd.tyAvl.bSeverity			:= TRUE;
//					tyNotificationSnd.tyAvl.bNotificationCode	:= TRUE;
//					tyNotificationSnd.tyAvl.bDescription		:= TRUE;
//					tyNotificationSnd.tyData.eSeverity			:= HermesSeverityError;
//					tyNotificationSnd.tyData.iNotificationCode	:= UDINT_TO_INT(udiStatus2);
//					tyNotificationSnd.tyData.sDescription		:= a_tyAlmText[udiStatus2].sAlmText;
//
//				END_IF
//
//			ELSE	//"Compare Type ID" Not Ticked
//
//				IF p_tyParam.bOverwrite THEN	//"Overwrite" Ticked
//
//					IF tyBoardAvailableRcv.tyAvl.bThickness AND tyBoardAvailableRcv.tyAvl.bTopClearanceHeight AND tyBoardAvailableRcv.tyAvl.bBottomClearanceHeight AND p_bBASltEn THEN	//Camparing Slot Parameters
//
//						udiStatus2	:= fHermesCmpSlt(tyBoardAvailableRcv.tyData.eFlippedBoard , tyBoardAvailableRcv.tyData.rThickness , tyBoardAvailableRcv.tyData.rTopClearanceHeight , tyBoardAvailableRcv.tyData.rBottomClearanceHeight , p_diMinSltValue , p_diMaxSltValue , p_diPitch , p_diSltToSltInUM , p_diTtlSlt);
//
//						IF udiStatus2 <> 0 THEN
//
//							bAccDataReq		:= TRUE;
//							bBABlkUS			:= TRUE;
//							bOverWriteSlt	:= TRUE;
//
//							fbGetSlt.eFlippedBrd				:= tyBoardAvailableRcv.tyData.eFlippedBoard;
//							fbGetSlt.rThicknessInMM				:= tyBoardAvailableRcv.tyData.rThickness;
//							fbGetSlt.rTopClearanceHeightInMM	:= tyBoardAvailableRcv.tyData.rTopClearanceHeight;
//							fbGetSlt.rBtmClearanceHeightInMM	:= tyBoardAvailableRcv.tyData.rBottomClearanceHeight;
//							fbGetSlt.diSltToSltInUM				:= p_diSltToSltInUM;
//							fbGetSlt.diTtlSlt					:= p_diTtlSlt;
//							fbGetSlt;
//
//							diReqMinSltValue	:= fbGetSlt.diMinSltValue;
//							diReqMaxSltValue	:= fbGetSlt.diMaxSltValue;
//							diReqPitch			:= fbGetSlt.diPitch;
//
//						END_IF
//
//					END_IF
//
//					IF tyBoardAvailableRcv.tyAvl.bWidth  AND p_bBAWidthEn (*AND p_usiLinkProdRcpCurrRcpMcMod = 0*) THEN	//Comparing Width Parameter
//						IF REAL_TO_DINT(tyBoardAvailableRcv.tyData.rWidth * 1000) <> p_diWidthInUM THEN
//
//							bAccDataReq		:= TRUE;
//							bBABlkUS			:= TRUE;
//							bOverWriteWidth	:= TRUE;
//
//							diReqWidthInUM	:= REAL_TO_DINT(tyBoardAvailableRcv.tyData.rWidth * 1000);
//
//						END_IF
//					END_IF
//
//				ELSE	//"Compare Type ID" Not Ticked and "Overwrite" Not Ticked, Error if not same
//
//					IF tyBoardAvailableRcv.tyAvl.bThickness AND tyBoardAvailableRcv.tyAvl.bTopClearanceHeight AND tyBoardAvailableRcv.tyAvl.bBottomClearanceHeight AND p_bBASltEn AND p_bRdyRcv THEN	//Camparing Slot Parameters
//						udiStatus2	:= fHermesCmpSlt(tyBoardAvailableRcv.tyData.eFlippedBoard , tyBoardAvailableRcv.tyData.rThickness , tyBoardAvailableRcv.tyData.rTopClearanceHeight , tyBoardAvailableRcv.tyData.rBottomClearanceHeight , p_diMinSltValue , p_diMaxSltValue , p_diPitch , p_diSltToSltInUM , p_diTtlSlt);
//
//						IF udiStatus2 <> 0 THEN
//
//							bBABlkUS		:= TRUE;
//
//							eStatus2	:= Error;
//
//							IF udiStatus2 = 2914 THEN
//								udiStatus2	:= 10120;	//Input First Slot Is Invalid
//							ELSIF udiStatus2 = 2915 THEN
//								udiStatus2	:= 10121;	//Input Last Slot Is Invalid
//							ELSIF udiStatus2 = 2916 THEN
//								udiStatus2	:= 10122;	//Input Pitch Is Invalid
//							ELSIF udiStatus2 = 2917 THEN
//								udiStatus2	:= 10123;	//Input Slot To Slot Distance Is Invalid
//							ELSIF udiStatus2 = 2918 THEN
//								udiStatus2	:= 10124;	//Input Total Slot Is Invalid
//							ELSIF udiStatus2 = 2919 THEN
//								udiStatus2	:= 10125;	//Input Thickness Is Invalid
//							ELSIF udiStatus2 = 2920 THEN
//								udiStatus2	:= 10126;	//Input Top Clearance Height Is Invalid
//							ELSIF udiStatus2 = 2921 THEN
//								udiStatus2	:= 10127;	//Input Bottom Clearance Height Is Invalid
//							ELSIF udiStatus2 = 2922 THEN
//								udiStatus2	:= 10128;	//Recipe First Slot Value & Board Available Data Not Match With Same Product Type Id
//							ELSIF udiStatus2 = 2923 THEN
//								udiStatus2	:= 10129;	//Recipe Last Slot Value & Board Available Data Not Match With Same Product Type Id
//							ELSIF udiStatus2 = 2924 THEN
//								udiStatus2	:= 10130;	//Recipe Pitch Value & Board Available Data Not Match With Same Product Type Id
//							END_IF
//
//							fHermesAddOneMsgSend(ADR(a_eMsgSend) , ADR(udiMsgSendBffr) , HermesMsgTypeNotification);
//
//							tyNotificationSnd.tyAvl.bSeverity			:= TRUE;
//							tyNotificationSnd.tyAvl.bNotificationCode	:= TRUE;
//							tyNotificationSnd.tyAvl.bDescription		:= TRUE;
//							tyNotificationSnd.tyData.eSeverity			:= HermesSeverityError;
//							tyNotificationSnd.tyData.iNotificationCode	:= UDINT_TO_INT(udiStatus2);
//							tyNotificationSnd.tyData.sDescription		:= a_tyAlmText[udiStatus2].sAlmText;
//
//						END_IF
//					END_IF
//
//					IF tyBoardAvailableRcv.tyAvl.bWidth AND p_bBAWidthEn AND p_bRdyRcv THEN	//Comparing Width Parameter
//						IF REAL_TO_DINT(tyBoardAvailableRcv.tyData.rWidth * 1000) <> p_diWidthInUM THEN
//
//							bBABlkUS		:= TRUE;
//
//							eStatus2	:= Error;
//							udiStatus2	:= 10131;	//Width Different With Same Product Type Id
//
//							fHermesAddOneMsgSend(ADR(a_eMsgSend) , ADR(udiMsgSendBffr) , HermesMsgTypeNotification);
//
//							tyNotificationSnd.tyAvl.bSeverity			:= TRUE;
//							tyNotificationSnd.tyAvl.bNotificationCode	:= TRUE;
//							tyNotificationSnd.tyAvl.bDescription		:= TRUE;
//							tyNotificationSnd.tyData.eSeverity			:= HermesSeverityError;
//							tyNotificationSnd.tyData.iNotificationCode	:= UDINT_TO_INT(udiStatus2);
//							tyNotificationSnd.tyData.sDescription		:= a_tyAlmText[udiStatus2].sAlmText;
//
//						END_IF
//					END_IF
//
//				END_IF
//
//			END_IF
//			                                                       //Add
//		ELSIF (p_bAccDataRdy = FALSE) OR bTransporting = TRUE THEN //AND p_bUIInsertBrdPrep = FALSE THEN
//
//			bAccDataReq		:= FALSE;
//			bBABlkUS		:= FALSE;
//			bOverWriteSlt	:= FALSE;
//			bOverWriteWidth	:= FALSE;
//
//		END_IF
//
//	ELSE
//
//		bAccDataReq		:= FALSE;
//		bBABlkUS		:= TRUE;
//		bOverWriteSlt	:= FALSE;
//		bOverWriteWidth	:= FALSE;
//
//	END_IF

END_ACTION
```

#### Act_Background_ChgConfig.st
```iecst
(** 2019-05-04 **)
ACTION Act_Background_ChgConfig:

	IF eStatus2 <> Error THEN

		IF (tyParamOld.iLaneID <> p_tyParam.iLaneID) OR (tyParamOld.sHostAddress <> p_tyParam.sHostAddress) OR (tyParamOld.uiHostPort <> p_tyParam.uiHostPort)
			OR (tyParamOld.bFeatureBoardForecast <> p_tyParam.bFeatureBoardForecast) OR (tyParamOld.bFeatureCheckAliveResponse <> p_tyParam.bFeatureCheckAliveResponse) OR (tyParamOld.bFeatureQueryBoardInfo <> p_tyParam.bFeatureQueryBoardInfo)
			OR (tyParamOld.bFeatureCommand <> p_tyParam.bFeatureCommand)
			THEN

			fHermesAddOneMsgSend(ADR(a_eMsgSend) , ADR(udiMsgSendBffr) , HermesMsgTypeNotification);

			tyNotificationSnd.tyAvl.bSeverity			:= TRUE;
			tyNotificationSnd.tyAvl.bNotificationCode	:= TRUE;
			tyNotificationSnd.tyAvl.bDescription		:= TRUE;
			tyNotificationSnd.tyData.eSeverity			:= HermesSeverityFatalError;
			tyNotificationSnd.tyData.iNotificationCode	:= 3;
			tyNotificationSnd.tyData.sDescription		:= 'Configuration Changed';

			bRstConnection	:= TRUE;

		END_IF

	END_IF

END_ACTION
```

#### Act_Background_ChkAlive.st
```iecst
(** 2019-05-30 **)
ACTION Act_Background_ChkAlive:

	IF eStatus1 <> Error THEN

		//Standard Check Alive (Without Ping & Pong)
		fbCheckAlive.bDataRcv		:= tyMsgTypeRcv.bCheckAlive OR tyMsgTypeRcv.bBoardAvailable OR tyMsgTypeRcv.bRevokeBoardAvailable OR tyMsgTypeRcv.bTransportFinished OR tyMsgTypeRcv.bTransportFinished OR tyMsgTypeRcv.bBoardForecast OR tyMsgTypeRcv.bSendBoardInfo OR tyMsgTypeRcv.bCommand ;
		fbCheckAlive.tSendTm		:= p_tyParam.tSndAlive;
		fbCheckAlive.tRcvTimeOut	:= p_tyParam.tRcvAlive;
		fbCheckAlive(bEn := TRUE);

		IF fbCheckAlive.udiStatus > 0 AND fbCheckAlive.udiStatus < 65534 THEN
			eStatus1	:= Error;

			IF fbCheckAlive.udiStatus = 2767 THEN
				udiStatus1	:= 10132;	//Check Alive Time Out
			ELSE
				udiStatus1	:= fbCheckAlive.udiStatus;
			END_IF

			fHermesAddOneMsgSend(ADR(a_eMsgSend) , ADR(udiMsgSendBffr) , HermesMsgTypeNotification);

			tyNotificationSnd.tyAvl.bSeverity			:= TRUE;
			tyNotificationSnd.tyAvl.bNotificationCode	:= TRUE;
			tyNotificationSnd.tyAvl.bDescription		:= TRUE;
			tyNotificationSnd.tyData.eSeverity			:= HermesSeverityFatalError;
			tyNotificationSnd.tyData.iNotificationCode	:= UDINT_TO_INT(udiStatus1);
			tyNotificationSnd.tyData.sDescription		:= a_tyAlmText[udiStatus1].sAlmText;

		ELSE
			IF EDGEPOS(fbCheckAlive.bDataSend) THEN
				fHermesAddOneMsgSend(ADR(a_eMsgSend) , ADR(udiMsgSendBffr) , HermesMsgTypeCheckAlive);
				tyCheckAliveSnd	:= fbCheckAlive.tyDataSend;
			END_IF

		END_IF

		tyMsgTypeRcv.bCheckAlive	:= FALSE;	//Reset Check Alive

	END_IF

END_ACTION
```

#### Act_Background_CmpParamRcv.st
```iecst
(** 2019-03-25 **)
ACTION Act_Background_CmpParamRcv:

	IF eStatus2 <> Error THEN

		IF tyMsgTypeRcv.bTransportFinished = TRUE THEN
			udiStatus2	:= fHermesChkParamSTTF(tyStartTransport , tyTransportFinished);

			IF udiStatus2 <> 0 THEN
				eStatus2	:= Error;

				IF udiStatus2 = 2714 THEN
					udiStatus2	:= 10104;	//BoardId Mismatch While Checking Start Transport & Transport Finished
				ELSIF udiStatus2 = 2715 THEN
					udiStatus2	:= 10105;	//BoardId Missing While Checking Start Transport & Transport Finished
				END_IF

				fHermesAddOneMsgSend(ADR(a_eMsgSend) , ADR(udiMsgSendBffr) , HermesMsgTypeNotification);

				tyNotificationSnd.tyAvl.bSeverity			:= TRUE;
				tyNotificationSnd.tyAvl.bNotificationCode	:= TRUE;
				tyNotificationSnd.tyAvl.bDescription		:= TRUE;
				tyNotificationSnd.tyData.eSeverity			:= HermesSeverityFatalError;
				tyNotificationSnd.tyData.iNotificationCode	:= UDINT_TO_INT(udiStatus2);
				tyNotificationSnd.tyData.sDescription		:= a_tyAlmText[udiStatus2].sAlmText;

			END_IF
		END_IF

		//SendBoardInfo
		IF tyServiceDescriptionRcv.tyAvl.tySupportedFeatures.bFeatureSendBoardInfo = TRUE AND p_tyParam.bFeatureQueryBoardInfo THEN
			IF tyMsgTypeRcv.bSendBoardInfo = TRUE THEN //AND p_bQueryBoardInfo THEN
				udiStatus2	:= fHermesChkParamSBIQBI(tySendBoardInfoRcv , tyQueryBoardInfo);

				IF udiStatus2 <> 0 THEN
					eStatus2	:= Error;

					IF udiStatus2 = 2769 THEN
						udiStatus2	:= 10170;	//Top Barcode Mismatch While Checking SendBoardInfo & QueryBoardInfo
					ELSIF udiStatus2 = 2770 THEN
						udiStatus2	:= 10171;	//Top Barcode Missing While Checking SendBoardInfo & QueryBoardInfo
					ELSIF udiStatus2 = 2771 THEN
						udiStatus2	:= 10172;	//Bottom Barcode Mismatch While Checking SendBoardInfo & QueryBoardInfo
					ELSIF udiStatus2 = 2772 THEN
						udiStatus2	:= 10173;	//Bottom Barcode Missing While Checking SendBoardInfo & QueryBoardInfo
					END_IF

					fHermesAddOneMsgSend(ADR(a_eMsgSend) , ADR(udiMsgSendBffr) , HermesMsgTypeNotification);

					tyNotificationSnd.tyAvl.bSeverity			:= TRUE;
					tyNotificationSnd.tyAvl.bNotificationCode	:= TRUE;
					tyNotificationSnd.tyAvl.bDescription		:= TRUE;
					tyNotificationSnd.tyData.eSeverity			:= HermesSeverityError;
					tyNotificationSnd.tyData.iNotificationCode	:= UDINT_TO_INT(udiStatus2);
					tyNotificationSnd.tyData.sDescription		:= a_tyAlmText[udiStatus2].sAlmText;

					tyMsgTypeRcv.bSendBoardInfo := FALSE; //reset, else will latching
				END_IF
			END_IF
		END_IF

		//check for route where reverse route, the board-id of forecast match with machine ready
		fHermesChkParamBFMR(tyBoardForecastRcv , tyMachineReady);

	END_IF

END_ACTION
```

#### Act_Background_Info.st
```iecst
(** 2020-09-10 **)
ACTION Act_Background_Info:
	IF usiAccDataStep <> 0 AND usiBFAccDataStep <> 0 THEN
		//Info Message for "BoardAvailable" and "BoardForecast"
		p_sInfoMsg		:= 'Upstream Hermes Request New Recipe';
		p_sInfoMsg		:= CONCAT(p_sInfoMsg , '$r$n');
		p_sInfoMsg		:= CONCAT(p_sInfoMsg , 'Old Recipe Name : ');
		p_sInfoMsg		:= CONCAT(p_sInfoMsg , p_sRecipeNm);
		p_sInfoMsg		:= CONCAT(p_sInfoMsg , '$r$n');
		p_sInfoMsg		:= CONCAT(p_sInfoMsg , 'Old Recipe Width : ');
		sWidthInUMTemp	:= DINT_TO_STRING(p_diWidthInUM / 1000);
		p_sInfoMsg		:= CONCAT(p_sInfoMsg , sWidthInUMTemp);
		p_sInfoMsg		:= CONCAT(p_sInfoMsg , '$r$n');
		p_sInfoMsg		:= CONCAT(p_sInfoMsg , 'New Recipe Name : ');
		p_sInfoMsg		:= CONCAT(p_sInfoMsg , sReqRecipeNm);
		p_sInfoMsg		:= CONCAT(p_sInfoMsg , '$r$n');
		p_sInfoMsg		:= CONCAT(p_sInfoMsg , 'New Recipe Width : ');
		sWidthInUMTemp	:= DINT_TO_STRING(diReqWidthInUM / 1000);
		p_sInfoMsg		:= CONCAT(p_sInfoMsg , sWidthInUMTemp);
	END_IF

	IF bRcvBoardInfoOk THEN
		//Info Message 1 for "SendBoardInfo"
		p_sInfoMsg1     := 'Board Info Received From Upstream';
		p_sInfoMsg1		:= CONCAT(p_sInfoMsg1 , '$r$n');
		p_sInfoMsg1		:= CONCAT(p_sInfoMsg1 , 'PCB Transfer to Last Zone is Blocked');
		p_sInfoMsg1		:= CONCAT(p_sInfoMsg1 , '$r$n');
		p_sInfoMsg1		:= CONCAT(p_sInfoMsg1 , 'Please Insert PCB to Last Zone Outlet');
		p_sInfoMsg1		:= CONCAT(p_sInfoMsg1 , '$r$n');
		p_sInfoMsg1		:= CONCAT(p_sInfoMsg1 , 'and PCB Data Will Be Overwritten');
		p_sInfoMsg1		:= CONCAT(p_sInfoMsg1 , '$r$n');
		p_sInfoMsg1		:= CONCAT(p_sInfoMsg1 , 'To Cancel,unpress the Query Board Info Button');
	END_IF

	IF bRcvBoardInfoIncompl THEN
		p_sInfoMsg2     := 'Board Info Not Found From Upstream';
	END_IF

END_ACTION
```

#### Act_Background_Log.st
```iecst
(** 2019-05-01 **)
ACTION Act_Background_Log:

	IF eStatus3 <> Error THEN

		IF udiWriteLogCntr <> udiLogCntr THEN

			CASE iWriteLogStep OF

				0:
					dtCurrDTTemp			:= p_dtCurrDT;
					fbFileAppend1.sFile		:= DT_TO_STRING(dtCurrDTTemp);
					fbFileAppend1.sFile		:= MID(fbFileAppend1.sFile , 10 , 4);
					fbFileAppend1.sFile		:= CONCAT('_' , fbFileAppend1.sFile);
					fbFileAppend1.sFile		:= CONCAT(p_sProgNm , fbFileAppend1.sFile);
					fbFileAppend1.sFile		:= CONCAT(fbFileAppend1.sFile , '.dat');

					fbFileAppend1.p_Src		:= ADR(a_sLogList[udiWriteLogCntr]);
					fbFileAppend1.udiLen	:= LEN(a_sLogList[udiWriteLogCntr]);

					iWriteLogStep	:= 1;

				1:
					fbFileAppend1(bEn := TRUE);
					IF fbFileAppend1.udiStatus = 0 THEN
						fbFileAppend1(bEn := FALSE);

						udiWriteLogCntr	:= udiWriteLogCntr + 1;
						IF udiWriteLogCntr = 11 THEN
							udiWriteLogCntr	:= 1;
						END_IF

						iWriteLogStep	:= 0;

					ELSIF fbFileAppend1.udiStatus < 65534 THEN
						eStatus3	:= Error;

						IF fbFileAppend1.udiStatus = 1900 THEN
							udiStatus3	:= 10148;	//File Open Error While Writing Log
						ELSIF fbFileAppend1.udiStatus = 1901 THEN
							udiStatus3	:= 10149;	//File Create Error While Writing Log
						ELSIF fbFileAppend1.udiStatus = 1913 THEN
							udiStatus3	:= 10150;	//Get File Info Error While Writing Log
						ELSIF fbFileAppend1.udiStatus = 1903 THEN
							udiStatus3	:= 10151;	//File Write Error While Writing Log
						ELSIF fbFileAppend1.udiStatus = 1904 THEN
							udiStatus3	:= 10152;	//File Close Error While Writing Log
						ELSIF fbFileAppend1.udiStatus = 1914 THEN
							udiStatus3	:= 10153;	//Directory Does Not Exist While Writing Log
						ELSE
							udiStatus3	:= fbFileAppend1.udiStatus;
						END_IF

						iWriteLogStep	:= 0;

					END_IF

			END_CASE

		END_IF

	END_IF

END_ACTION
```

#### Act_Background_ProcessData.st
```iecst
(** 2023-08-01 **)
ACTION Act_Background_ProcessData:

	//update from event to trigger message externally

	//when stop transport, Svy send board arrived , prompt send no board id forecast
	bStopTransportSnd := EDGEPOS (fbSequenceUS.eMsgTypeSnd = HermesMsgTypeStopTransport) AND p_bConvHvBrd ; //Incoming Zone have board;

	IF bStopTransportSnd THEN
		tyBoardArrivedInfo := tyBoardAvailableRcv;
	END_IF

END_ACTION
```
